		(* Menu war aktiv -> Escape -> Menu deaktivieren *)
	ELSIF (Xus_TN_MENU.in_State = INT#02) THEN
		us_TN_MENU_POPUP.bo_Destroy := TRUE;
		Xus_TN_MENU.bo_Update := TRUE;
		Xus_TN_MENU.in_State := INT#01;
		bo_Reset_Position := TRUE;

		Xus_TN_SCREEN.bo_Menue_Bar_Dialog := FALSE;
	END_IF;
END_IF;

(* Menu aktiv *)
IF (Xus_TN_MENU.in_State = INT#02) THEN

	(* Return *)
	IF (by_New_KeyCode = BYTE#13)  THEN
		us_TN_MENU_POPUP.bo_Destroy := TRUE;
		Xus_TN_MENU.bo_Update := TRUE;
		Xus_TN_MENU.in_State := INT#01;
		bo_Reset_Position := TRUE;
		Xus_TN_MENU.in_Menu_Selected := (Xus_TN_MENU.in_Cur_Menu_Item * INT#10) + Xus_TN_MENU.in_Cur_Sub_Item;
		Xus_TN_SCREEN.by_Input_Exten_Code := BYTE#00;

		Xus_TN_SCREEN.bo_Menue_Bar_Dialog := FALSE;

		(* Destroy-Befehl -> Popup-Menu beenden *)
	ELSIF (Xus_TN_MENU.bo_Destroy = TRUE) THEN
		us_TN_MENU_POPUP.bo_Destroy := TRUE;
		Xus_TN_MENU.bo_Update := TRUE;
		Xus_TN_MENU.in_State := INT#01;
		bo_Reset_Position := TRUE;
		Xus_TN_MENU.in_Menu_Selected := INT#00;
		Xus_TN_SCREEN.by_Input_Exten_Code := BYTE#00;

		Xus_TN_SCREEN.bo_Menue_Bar_Dialog := FALSE;

	END_IF;

	IF (by_New_KeyCode = BYTE#67) THEN (* Cursor rechts *)
		in_Scroll_Offset := INT#1;
		Xus_TN_MENU.bo_Update := TRUE;
		Xus_TN_SCREEN.by_Input_Exten_Code := BYTE#00;

	ELSIF (by_New_KeyCode = BYTE#68) THEN (* Cursor links *)
		in_Scroll_Offset := -1;
		Xus_TN_MENU.bo_Update := TRUE;
		Xus_TN_SCREEN.by_Input_Exten_Code := BYTE#00;
	END_IF;
END_IF;

IF bo_Reset_Position = TRUE THEN
	bo_Reset_Position := FALSE;
	Xus_TN_MENU.in_X_SM_old := -1;
	Xus_TN_MENU.in_Y_SM_old := -1;
	Xus_TN_MENU.in_X_SM_new := -1;
	Xus_TN_MENU.in_Y_SM_new := -1;
END_IF;

(* POPUP-Menu updaten *)
IF (Xus_TN_MENU.in_State > INT#00) AND (Xus_TN_MENU.bo_Update = TRUE) THEN

	Xus_TN_MENU.bo_Update := FALSE; 

	in_ROW := Xus_TN_MENU.in_Y;
	in_COL := Xus_TN_MENU.in_X;

	(* Scrolloffset *)
	IF in_Scroll_Offset <> INT#00 THEN
		Xus_TN_MENU.in_Cur_Menu_Item := INC2(Xus_TN_MENU.in_Cur_Menu_Item,in_Scroll_Offset,1,Xus_TN_MENU.in_Menu_E_Count);
		in_Scroll_Offset := INT#00;
	ELSE
		(* Item = 0 und kein Scrolloffset *)
		IF (Xus_TN_MENU.in_Cur_Menu_Item = INT#00) THEN
			Xus_TN_MENU.in_Cur_Menu_Item := INT#01;
		END_IF;
	END_IF;

	(* alle Menutext zeichnen *)
	FOR in_Count := INT#01 TO Xus_TN_MENU.in_Menu_E_Count DO;

		(* Zeichenfarbe bestimmen *)
		IF (in_Count = Xus_TN_MENU.in_Cur_Menu_Item) AND (Xus_TN_MENU.in_State > INT#01 ) THEN
			by_ATTR := Xus_TN_MENU.by_Attr_mF;

			Xus_TN_MENU.in_Y_SM_new := in_ROW + INT#01;
			Xus_TN_MENU.in_X_SM_new := in_COL;

		ELSE
			by_ATTR := Xus_TN_MENU.by_Attr_oF;
		END_IF;

		st_MENU_TITLE := ELEMENT_GET(SEP:=BYTE#35,POS:=in_Count - 1,ELEMENT:=st_MENU_BAR);

		in_TITLE_Length := LEN(st_MENU_TITLE) + INT#02;

		FB_TN_SC_WRITE_C(	Iin_Y := in_ROW,
							Iin_X := in_COL,
							Iby_ATTR := by_ATTR,
							Iin_LENGTH := in_TITLE_Length,
							Iin_OPTION := INT#02,
							Ist_STRING := st_MENU_TITLE,
							Xus_TN_SCREEN := Xus_TN_SCREEN);

		in_COL := in_COL + in_TITLE_Length;

	END_FOR;
END_IF;

IF Xus_TN_MENU.in_X_SM_new <> Xus_TN_MENU.in_X_SM_old THEN

	(* SubMenu ist aktiv -> beenden                                     *)
	IF us_TN_MENU_POPUP.bo_Activ = TRUE THEN
		us_TN_MENU_POPUP.bo_Destroy := TRUE;

		(* Sub-Menu bearbeiten *)
		FB_TN_INPUT_MENU_POPUP(	Xus_TN_MENU_POPUP := us_TN_MENU_POPUP,
								Xus_TN_SCREEN := Xus_TN_SCREEN);
	END_IF;

	IF us_TN_MENU_POPUP.bo_Activ = FALSE THEN
		(* Popup-Menu zu aktuellen Menu parametrieren und ausführen         *)
		in_Index := Xus_TN_MENU.in_Cur_Menu_Item;

		us_TN_MENU_POPUP.in_Y := Xus_TN_MENU.in_Y_SM_new;
		us_TN_MENU_POPUP.in_X := Xus_TN_MENU.in_X_SM_new;
		us_TN_MENU_POPUP.by_Attr_mF := Xus_TN_MENU.by_Attr_mF;
		us_TN_MENU_POPUP.by_Attr_oF := Xus_TN_MENU.by_Attr_oF;
		us_TN_MENU_POPUP.st_Menu_Text := ELEMENT_GET(SEP:=BYTE#37,POS:=in_Index,ELEMENT:=Xus_TN_MENU.st_MENU_TEXT);
		us_TN_MENU_POPUP.bo_Create := TRUE;

		Xus_TN_MENU.in_X_SM_old := Xus_TN_MENU.in_X_SM_new;
		Xus_TN_MENU.in_Y_SM_old := Xus_TN_MENU.in_Y_SM_new;

	END_IF;
END_IF;

(* Popup-Menu zyklisch aufrufen *)
FB_TN_INPUT_MENU_POPUP(	Xus_TN_MENU_POPUP := us_TN_MENU_POPUP,
						Xus_TN_SCREEN := Xus_TN_SCREEN);

(* aktuelles Item vom Popup-Menu kopieren *)
Xus_TN_MENU.in_Cur_Sub_Item := us_TN_MENU_POPUP.in_Cur_Item;

(* Destroy-Befehl *)
IF (Xus_TN_MENU.in_State = INT#01) THEN
	IF (Xus_TN_MENU.bo_Destroy = TRUE) THEN
		Xus_TN_MENU.in_State := INT#00;
		Xus_TN_MENU.bo_Destroy := FALSE;
		Xus_TN_MENU.in_Cur_Menu_Item := INT#00;
		Xus_TN_MENU.in_Cur_Sub_Item := INT#00;
	END_IF;
END_IF;

(* revision history
ks	06. apr. 2011	rev 1.1
	list_len und list_get durch element_count und element_get ersetzt

ks	10. mai. 2010	rev 1.0
	original version
*)

END_FUNCTION_BLOCK

// ---- POUs/TELNET_VISION/TN_RECEIVE.TcPOU
FUNCTION_BLOCK TN_RECEIVE
VAR_IN_OUT
	R_BUF :	NETWORK_BUFFER;
	Xus_TN_SCREEN : us_TN_SCREEN;
END_VAR
VAR
	REQ_Size : UINT;
	REQ1 : BYTE;
	REQ2 : BYTE;
	REQ3 : BYTE;
END_VAR

(*
version 1.0		10. mai 2010
programmer		ks
tested by		ks

TN_RECEIVE empfängt Tastatureingaben vom Telnet Client und wertet diese aus
*)

(* Datenempfang auswertung *)
Xus_TN_SCREEN.by_Input_ASCII_Code := BYTE#00;
Xus_TN_SCREEN.by_Input_Exten_Code := BYTE#00;

IF R_BUF.SIZE > UINT#0 THEN
	(* empfangene Daten auswerten *)
	REQ_Size := R_BUF.SIZE;
	REQ1 := R_BUF.BUFFER[0];
	REQ2 := R_BUF.BUFFER[1];
	REQ3 := R_BUF.BUFFER[2];

	IF REQ1 = BYTE#27 AND REQ_Size >= UINT#3 THEN (* Escape *)
		IF REQ2 = BYTE#91 THEN (* Cursor code *)
			IF (REQ3 >= BYTE#65 AND REQ3 <= BYTE#68) OR (REQ3 = BYTE#72) OR (REQ3 = BYTE#75) THEN (* 65..68 = Cursor o,u,r,l / 72 = POS1 / 75 = ENDE *)
				Xus_TN_SCREEN.by_Input_Exten_Code := REQ3;
			END_IF;
		ELSIF REQ2 = BYTE#79 THEN (* Sondertasten F1/F2/F3/F4 *)
			IF REQ3 >= BYTE#80 AND REQ3 <= BYTE#83 THEN
				Xus_TN_SCREEN.by_Input_Exten_Code := REQ3;
			END_IF;
		END_IF;
	ELSIF REQ1 >= BYTE#32 AND REQ1 <= BYTE#126 THEN
		Xus_TN_SCREEN.by_Input_ASCII_Code := REQ1;
		Xus_TN_SCREEN.bo_Input_ASCII_IsNum := ISC_NUM(REQ1); (* Auswertung auf Zahleneingabe *)
	ELSIF REQ1 = BYTE#8 OR REQ1 = BYTE#9 OR REQ1 = BYTE#13 OR REQ1 = BYTE#27 THEN (* prüfe auf Steuerzeichen 8=Backspace / 9=Tabulator / 13=Return / 27=Escape *)
		Xus_TN_SCREEN.by_Input_Exten_Code := REQ1;
	END_IF;

	(* Empfangsbuffer Datenlänge null eintragen (Telegramm zerstören *)
	R_BUF.SIZE := UINT#00;
END_IF;

(* revision history
ks	10. mai. 2010	rev 1.0
	original version
*)

END_FUNCTION_BLOCK

// ---- POUs/TELNET_VISION/TN_SEND_ROWS.TcPOU
FUNCTION_BLOCK TN_SEND_ROWS
VAR_IN_OUT
	IP_C : IP_C;
	S_BUF : NETWORK_BUFFER;
	Xus_TN_SCREEN : us_TN_SCREEN;
END_VAR
VAR_INPUT
	S_BUF_SIZE : INT;
END_VAR
VAR
	in_Line_Count : INT;(*Zähler um max alle 24 Zeilen zu durchlaufen*)
	in_Col_Count : INT;
	in_Last_Row_Index : INT;
	bo_Break_Loop : BOOL;
	in_Row_Count : INT;
	in_Offset : INT;
	in_Write_Index : INT;
	in_Write_Index_Backup : INT;
	by_Cur_Color : BYTE;
	by_last_Color : BYTE;
	in_Write_Stop : INT;
END_VAR

(*
version 1.0		10. mai 2010
programmer		ks
tested by		ks

TN_SEND_ROWS prüft den Bildschirmspeicher auf änderungen, und sendet diese zeilenweise an den Telnet Client 
*)

(* Verbindung vorhanden und kein Datensenden aktiv *)
IF (IP_C.C_STATE < BYTE#127 OR S_BUF.SIZE > UINT#0) THEN
	RETURN; (* nein -> Baustein beenden *)
END_IF;

(* aktuellen Schreibindex laden *)
in_Write_Index := UINT_TO_INT(S_BUF.SIZE) - 1;

(* aktuellen Schreibindex zwischenspeichern *)
in_Write_Index_Backup := in_Write_Index;

(* positive Flanke Connect on *)
IF (IP_C.C_STATE = BYTE#254) OR (Xus_TN_SCREEN.bo_Clear_Screen) THEN

	(* Clear-Screen Meldung rücksetzen *)
	Xus_TN_SCREEN.bo_Clear_Screen := FALSE;

	(* alle Zeilen für Update markieren *)
	FOR in_Line_Count := INT#00 TO INT#23 DO
		Xus_TN_SCREEN.bya_Line_Update[in_Line_Count] := TRUE;
	END_FOR;

	(* ESC [0;30,40m  Reset Attributes + Black,Black *)
	in_Write_Index := in_Write_Index + INT#1;
	S_BUF.BUFFER[in_Write_Index] := BYTE#16#1B; (* ESC *)
	in_Write_Index := in_Write_Index + INT#1;
	S_BUF.BUFFER[in_Write_Index] := BYTE#16#5B; (* [ *)
	in_Write_Index := in_Write_Index + INT#1;
	S_BUF.BUFFER[in_Write_Index] := BYTE#16#30; (* 0 *)
	in_Write_Index := in_Write_Index + INT#1;
	S_BUF.BUFFER[in_Write_Index] := BYTE#16#3B; (* ; *)
	in_Write_Index := in_Write_Index + INT#1;
	S_BUF.BUFFER[in_Write_Index] := BYTE#16#33; (* 3 *)

	(* Einerstelle Farbe Foreground ausgeben *)
	in_Write_Index := in_Write_Index + INT#1;
	S_BUF.BUFFER[in_Write_Index] := (SHR(Xus_TN_SCREEN.by_Clear_Screen_Attr,4) OR BYTE#16#30);

	in_Write_Index := in_Write_Index + INT#1;
	S_BUF.BUFFER[in_Write_Index] := BYTE#16#3B; (* ; *)
	in_Write_Index := in_Write_Index + INT#1;
	S_BUF.BUFFER[in_Write_Index] := BYTE#16#34; (* 4 *)

	(* Einerstelle Farbe Background ausgeben *)
	in_Write_Index := in_Write_Index + INT#1;
	S_BUF.BUFFER[in_Write_Index] := ((Xus_TN_SCREEN.by_Clear_Screen_Attr AND BYTE#16#07) OR BYTE#16#30);

	in_Write_Index := in_Write_Index + INT#1;
	S_BUF.BUFFER[in_Write_Index] := BYTE#16#6D; (* m *)

	(* ESC[2J Clear screen and home cursor *)
	in_Write_Index := in_Write_Index + INT#1;
	S_BUF.BUFFER[in_Write_Index] := BYTE#16#1B; (* ESC *)
	in_Write_Index := in_Write_Index + INT#1;
	S_BUF.BUFFER[in_Write_Index] := BYTE#16#5B; (* [ *)
	in_Write_Index := in_Write_Index + INT#1;
	S_BUF.BUFFER[in_Write_Index] := BYTE#16#32; (* 2 *)
	in_Write_Index := in_Write_Index + INT#1;
	S_BUF.BUFFER[in_Write_Index] := BYTE#16#4A; (* J *)

	(* ESC [?7l Off *)
	in_Write_Index := in_Write_Index + INT#1;
	S_BUF.BUFFER[in_Write_Index] := BYTE#16#1B; (* ESC *)
	in_Write_Index := in_Write_Index + INT#1;
	S_BUF.BUFFER[in_Write_Index] := BYTE#16#5B; (* [ *)
	in_Write_Index := in_Write_Index + INT#1;
	S_BUF.BUFFER[in_Write_Index] := BYTE#16#3F; (* ? *)
	in_Write_Index := in_Write_Index + INT#1;
	S_BUF.BUFFER[in_Write_Index] := BYTE#16#37; (* 7 *)
	in_Write_Index := in_Write_Index + INT#1;
	S_BUF.BUFFER[in_Write_Index] := BYTE#16#6C; (* l *)

END_IF;

in_Last_Row_Index := INT#0;
bo_Break_Loop := FALSE;
in_Write_Stop := S_BUF_SIZE - 20;

(* alle Zeilen durchlaufen *)
FOR in_Line_Count := 0 TO 23 DO

	in_Offset := in_Row_Count * INT#80;

	(* prüfen ob Update einer Zeile notwendig ist bzw. nach Reconnect *)
	IF (Xus_TN_SCREEN.bya_Line_Update[in_Row_Count] = TRUE) THEN

		(* Schreib-Cursor positionieren *)
		in_Write_Index := in_Write_Index + INT#1;
		S_BUF.BUFFER[in_Write_Index] := BYTE#16#1B; (* ESC *)
		in_Write_Index := in_Write_Index + INT#1;
		S_BUF.BUFFER[in_Write_Index] := BYTE#16#5B; (* [ *)

		(* Zehnerstelle Zeilennummer ausgeben *)
		in_Write_Index := in_Write_Index + INT#1;
		S_BUF.BUFFER[in_Write_Index] :=
		SHR(INT_TO_BCDC(in_Row_Count + INT#1),INT#4) OR BYTE#16#30;

		(* Einerstelle Zeilennummer ausgeben *)
		in_Write_Index := in_Write_Index + INT#1;
		S_BUF.BUFFER[in_Write_Index] :=
		(INT_TO_BCDC(in_Row_Count + INT#1) AND BYTE#16#0F) OR BYTE#16#30;

		in_Write_Index := in_Write_Index + INT#1;
		S_BUF.BUFFER[in_Write_Index] := BYTE#16#3B; (* ; *)
		in_Write_Index := in_Write_Index + INT#1;
		S_BUF.BUFFER[in_Write_Index] := BYTE#16#31; (* 1 *)
		in_Write_Index := in_Write_Index + INT#1;
		S_BUF.BUFFER[in_Write_Index] := BYTE#16#48; (* H *)

		(* alle Spalten einer Zeile durchlaufen *)
		FOR in_Col_Count := 0 TO 79 DO

			(* aktuelle Farbe bestimmen *)
			by_Cur_Color := Xus_TN_SCREEN.bya_COLOR[in_Offset];
			IF (by_Cur_Color <> by_last_Color) OR (in_Col_Count = INT#00) THEN

				(* Farbeinstellung: ANSI-Sequenz ESC[X;Y;Zm ausgeben *)
				in_Write_Index := in_Write_Index + INT#1;
				S_BUF.BUFFER[in_Write_Index] := BYTE#16#1B; (* ESC *)

				in_Write_Index := in_Write_Index + INT#1;
				S_BUF.BUFFER[in_Write_Index] := BYTE#16#5B; (* [ *)

				(* Farbeinstellung: dunkel oder Hell und blinken bestimmen *)

					IF (((by_Cur_Color AND BYTE#2#10001000) XOR (by_last_Color AND BYTE#2#10001000)) <> BYTE#00) OR (in_Col_Count = 0) THEN

						in_Write_Index := in_Write_Index + INT#1;
						S_BUF.BUFFER[in_Write_Index] := BYTE#16#30; (* 0 *)
						in_Write_Index := in_Write_Index + INT#1;
						S_BUF.BUFFER[in_Write_Index] := BYTE#16#3B; (* ; *)

						(* keine dunklen Farben gewünscht -> dann Bold & Bright *)
						IF (by_Cur_Color AND BYTE#2#00001000) = BYTE#2#00000000 THEN

							(* auf Bold & Btight Farben umstellen *)
							in_Write_Index := in_Write_Index + INT#1;
							S_BUF.BUFFER[in_Write_Index] := BYTE#16#31; (* 1 *) 
							in_Write_Index := in_Write_Index + INT#1;
							S_BUF.BUFFER[in_Write_Index] := BYTE#16#3B; (* ; *)

						END_IF;

						(* blinkenden Farben gewünscht *)
						IF (by_Cur_Color AND BYTE#2#10000000) = BYTE#2#10000000 THEN 

							(* auf Bold & Bright Farben umstellen *)
							in_Write_Index := in_Write_Index + INT#1;
							S_BUF.BUFFER[in_Write_Index] := BYTE#16#35; (* 5 *) 
							in_Write_Index := in_Write_Index + INT#1;
							S_BUF.BUFFER[in_Write_Index] := BYTE#16#3B; (* ; *)

						END_IF;

					END_IF;

					(* Zehnerstelle Farbe Foreground ausgeben *)
					in_Write_Index := in_Write_Index + INT#1;
					S_BUF.BUFFER[in_Write_Index] := BYTE#16#33; (* 3 *)

					(* Einerstelle Farbe Foreground ausgeben *)
					in_Write_Index := in_Write_Index + INT#1;
					S_BUF.BUFFER[in_Write_Index] := ((SHR(by_Cur_Color,4) AND BYTE#2#00000111) OR BYTE#16#30);

					in_Write_Index := in_Write_Index + INT#1;
					S_BUF.BUFFER[in_Write_Index] := BYTE#16#3B; (* ; *)

					(* Zehnerstelle Farbe Background ausgeben *)
					in_Write_Index := in_Write_Index + INT#1;
					S_BUF.BUFFER[in_Write_Index] := BYTE#16#34; (* 4 *)

					(* Einerstelle Farbe Background ausgeben *)
					in_Write_Index := in_Write_Index + INT#1;
					S_BUF.BUFFER[in_Write_Index] := ((by_Cur_Color AND BYTE#2#00000111) OR BYTE#16#30); 

					in_Write_Index := in_Write_Index + INT#1;
					S_BUF.BUFFER[in_Write_Index] := BYTE#16#6D; (* m *)

					(* neue Farbe als letzt verwendete speichern *)
					by_last_Color := by_Cur_Color;

				END_IF;

				(* Buffer Ende vorzeitig erreicht -> Ende *)
				IF (in_Write_Index > in_Write_Stop) THEN

					bo_Break_Loop := TRUE;
					EXIT;

				END_IF;

				(* ein TEXT-Zeichen von Screenbuffer in den Sendebuffer übertragen *)
				in_Write_Index := in_Write_Index + INT#1;
				S_BUF.BUFFER[in_Write_Index] := Xus_TN_SCREEN.bya_CHAR[in_Offset];

				(* nächste Spalte anwählen *)
				in_Offset := in_Offset + INT#01;
			END_FOR;

			IF (bo_Break_Loop = TRUE) THEN;

				(* Buffer Ende vorzeitig erreicht -> nur bis zur letzten kompletten Zeile uebertragen *)
				in_Write_Index := in_Last_Row_Index;

				EXIT;
			END_IF;

			(* Buffer ist noch nicht voll -> neue Zeile ubernehmen *)
			in_Last_Row_Index := in_Write_Index;
			Xus_TN_SCREEN.bya_Line_Update[in_Row_Count] := FALSE;

		END_IF;

		(* naechste Zeile adressieren *)
		in_Row_Count := in_Row_Count + INT#01;

		(* ab letzter Zeile wieder von vorne beginnen *)
		IF (in_Row_Count > INT#23) THEN
			in_Row_Count := INT#00;
		END_IF;
		(*-----------------------------------------------*)


	END_FOR;

	(* wenn in einen Update-Zyklus alle Zeilen auf einmal geschafft wurden *)
	(* wird der Row_Count auf ersten Zeile gestellt *)
	(* soll das hässliche Grafikflackern verhindern *)
	(* ansonsten wird bei der letzen Zeile weitergemacht *)
	IF (bo_Break_Loop = FALSE) THEN
		in_Row_Count := INT#00;
	END_IF;

	(* Edit-Cursor positionieren *)
	IF (in_Write_Index <> in_Write_Index_Backup) THEN

		in_Write_Index := in_Write_Index + INT#1;
		S_BUF.BUFFER[in_Write_Index] := BYTE#16#1B; (* ESC *)
		in_Write_Index := in_Write_Index + INT#1;
		S_BUF.BUFFER[in_Write_Index] := BYTE#16#5B; (* [ *)

		(* Zehnerstelle Zeilennummer ausgeben *)
		in_Write_Index := in_Write_Index + INT#1;
		S_BUF.BUFFER[in_Write_Index] := SHR(INT_TO_BCDC(Xus_TN_SCREEN.in_Cursor_Y + 1),INT#4) OR BYTE#16#30;

		(* Einerstelle Zeilennummer ausgeben *)
		in_Write_Index := in_Write_Index + INT#1;
		S_BUF.BUFFER[in_Write_Index] := (INT_TO_BCDC(Xus_TN_SCREEN.in_Cursor_Y + 1) AND BYTE#16#0F) OR BYTE#16#30;

		in_Write_Index := in_Write_Index + INT#1;
		S_BUF.BUFFER[in_Write_Index] := BYTE#16#3B; (* ; *)

		(* Zehnerstelle Spaltenummer ausgeben *)
		in_Write_Index := in_Write_Index + INT#1;
		S_BUF.BUFFER[in_Write_Index] := SHR(INT_TO_BCDC(Xus_TN_SCREEN.in_Cursor_X + 1),INT#4) OR BYTE#16#30;

		(* Einerstelle Spaltennummer ausgeben *)
		in_Write_Index := in_Write_Index + INT#1;
		S_BUF.BUFFER[in_Write_Index] := (INT_TO_BCDC(Xus_TN_SCREEN.in_Cursor_X + 1) AND BYTE#16#0F) OR BYTE#16#30;

		in_Write_Index := in_Write_Index + INT#1;
		S_BUF.BUFFER[in_Write_Index] := BYTE#16#48; (* H *)

END_IF;

(* aktuellen Schreibindex speichern -> Senden anstossen *)
S_BUF.SIZE := TO_UINT(in_Write_Index + 1);

(* revision history
ks	10. mai. 2010	rev 1.0
	original version
*)

END_FUNCTION_BLOCK

// ---- POUs/NETWORK/LOG_VIEWPORT.TcPOU
FUNCTION_BLOCK LOG_VIEWPORT
VAR_IN_OUT
	LC : LOG_CONTROL;
	LV : us_LOG_VIEWPORT;
END_VAR
VAR
	pos : INT;
	count : INT;
	idx : INT;
	base : INT;
	update_pos : BOOL;
END_VAR

(*
version 1.0		01 mai 2010
programmer		ks
tested BY		ks

LOG_VIEWPORT erzeugt einen Liste der Meldungen des Loggingbuffers die innerhalb einer virtuellen Ansicht enthalten sind.
*)

(* Scroll Button verarbeiten *)
IF LV.MOVE_TO_X <> 0 THEN
	CASE LV.MOVE_TO_X OF
	30000: pos := 1 ; (* älteste Meldung anzeigen *)
	30001: pos := LC.SIZE; (* neueste Meldung anzeigen *)
	30002: pos := pos + LV.COUNT; (* eine Seite nach unten blättern -> Richtung neuere Nachrichten *)
	30003: pos := pos - LV.COUNT; (* eine Seite nach oben blättern -> Richtung ältere Nachrichten *)
	ELSE
		pos := pos + LV.MOVE_TO_X;
	END_CASE;
	update_pos := TRUE;
	LV.MOVE_TO_X := 0;
END_IF;

IF (LV.UPDATE_COUNT <> LC.UPDATE_COUNT) OR update_pos THEN (* Aktualisierung überwachen *)
	LV.UPDATE := TRUE;
	LV.UPDATE_COUNT := LC.UPDATE_COUNT;
	update_pos := FALSE;

	(* pos prüfen und übernehmen *)
	IF LC.RING_MODE THEN
		pos := LIMIT(1,pos,LC.SIZE - LV.COUNT + 1);
	ELSE
		IF LC.IDX > LV.COUNT THEN
			pos := LIMIT(1,pos,LC.IDX - LV.COUNT + 1);
		ELSE
			pos := 1;
		END_IF;
	END_IF;

	(* idxBasis berechnen *)
	base := LC.IDX - pos - LV.COUNT + 1;
	IF LC.RING_MODE THEN 
		(* Anzeige im Ringpuffermodus *)
		FOR count:= 1 TO LV.COUNT DO
			idx := base + count;
			IF idx < 1 THEN
				idx := idx + LC.SIZE;
			END_IF;
		END_FOR;
	ELSE
		(* Anzeige im Normalmodus *)
		FOR count:= 1 TO LV.COUNT DO
			idx := base + count;
			IF idx < 1 THEN
				(* Leere Zeile ausgeben *)
				LV.LINE_ARRAY[count] := 0;
			ELSE
				LV.LINE_ARRAY[count] := idx;
			END_IF;
		END_FOR;
	END_IF;
END_IF;

(* revision history
ks	01. mai 2010	rev 1.0
	original version
*)

END_FUNCTION_BLOCK

// ---- POUs/TELNET_VISION/TN_SC_VIEWPORT.TcPOU
FUNCTION_BLOCK TN_SC_VIEWPORT
VAR
	FB_TN_SC_WRITE : TN_SC_WRITE;
	FB_TON : TON;
END_VAR
VAR
	in_index : INT;
	in_Color : INT;
	by_Attr : BYTE;
	in_count : INT;
END_VAR
VAR_IN_OUT
	Xus_LOG_VIEWPORT : us_LOG_VIEWPORT;
	Xus_LOG_CONTROL : LOG_CONTROL;
	Xus_TN_SCREEN : us_TN_SCREEN;
END_VAR
VAR_INPUT
	Iin_X : INT;
	Iin_Y : INT;
	Iin_Width : INT;
	Idw_ATTR_1 : DWORD;
	Idw_ATTR_2 : DWORD;
	Iti_TIME : TIME;
END_VAR

(*
version 1.0		10. mai 2010
programmer		ks
tested by		ks

TN_SC_VIEWPORT verwaltet und zeichnet einen rechteckigen Bereich in dem der Log-buffer angezeigt wird
*)

(* LOG-Messages ausgeben *)

IF Xus_LOG_VIEWPORT.UPDATE AND FB_TON.Q THEN (* Update gewünscht und Verzögerungszeit abgelaufen *)
	Xus_LOG_VIEWPORT.UPDATE := FALSE;
	FOR in_count := 1 TO Xus_LOG_VIEWPORT.COUNT DO (* Alle Viewport-Zeilen abarbeiten *)
		in_index := Xus_LOG_VIEWPORT.LINE_ARRAY[in_count];
		(* Farbe aus den Option-Parameter auslesen >0,Level,Back,Front< *)
		in_Color := DWORD_TO_INT(Xus_LOG_CONTROL.MSG_OPTION[in_index] AND DWORD#2#1111);

		CASE in_Color OF
		0..3: by_Attr := BYTE_OF_DWORD(Idw_ATTR_1,INT_TO_BYTE(in_Color));
		4..7: by_Attr := BYTE_OF_DWORD(Idw_ATTR_2,INT_TO_BYTE(in_Color));
		ELSE
			by_Attr := BYTE_OF_DWORD(Idw_ATTR_1,BYTE#0);
		END_CASE;

		(* Message (Text + Farbe) ausgeben *)
		FB_TN_SC_WRITE(	Iin_Y := Iin_Y + in_count - INT#01,
						Iin_X := Iin_X,
						Iby_ATTR := by_Attr,
						Ist_STRING := FIX(str := Xus_LOG_CONTROL.MSG[in_index], L := Iin_Width, C := BYTE#32, M := INT#00), (* String rechts ergänzen bzw. kürzen *)
						Xus_TN_SCREEN := Xus_TN_SCREEN);

	END_FOR;

	(* Timer stoppen/rücksetzen *)
	FB_TON.IN := FALSE;
	FB_TON.PT := Iti_TIME;
	FB_TON();

END_IF;

(* Update-Zeitverzoegerung *)
FB_TON.IN := TRUE;
FB_TON.PT := Iti_TIME;
FB_TON();

(* revision history
ks	10. mai. 2010	rev 1.0
	original version
*)

END_FUNCTION_BLOCK

// ---- POUs/DEMO/TN_VISION_DEMO_2.TcPOU
PROGRAM TN_VISION_DEMO_2
VAR
	FB_TN_FRAMEWORK : TN_FRAMEWORK;
	FB_TN_SC_FILL : TN_SC_FILL;
	FB_TN_SC_WRITE_C : TN_SC_WRITE_C;
	FB_TN_SC_WRITE : TN_SC_WRITE;
	Xus_TN_MENU : us_TN_MENU;
	Xus_TN_INPUT_CONTROL : us_TN_INPUT_CONTROL;
	Xus_TN_SCREEN : us_TN_SCREEN;
	S_BUF : NETWORK_BUFFER;
	R_BUF : NETWORK_BUFFER;
	IP_C : IP_C;
END_VAR

FB_TN_FRAMEWORK(
	us_TN_INPUT_CONTROL := Xus_TN_INPUT_CONTROL ,
	us_TN_SCREEN := Xus_TN_SCREEN ,
	us_TN_MENU := Xus_TN_MENU ,
	S_BUF := S_BUF ,
	R_BUF:= R_BUF ,
	IP_C:= IP_C );

(* Initialisierung der Daten und Strukturen *)
IF (Xus_TN_SCREEN.in_Page_Number = INT#00) THEN
	Xus_TN_SCREEN.in_Page_Number := INT#01;

	(* Clear-Screen (Farbe setzen + Display löschen) *)
	Xus_TN_SCREEN.by_Clear_Screen_Attr := BYTE#16#00;
	Xus_TN_SCREEN.bo_Clear_Screen := TRUE;

	(* Screen initialisieren (mit Leerzeichen füllen) *)
	FB_TN_SC_FILL(	Iin_X1 := INT#00,
					Iin_Y1 := INT#00,
					Iin_X2 := INT#79,
					Iin_Y2 := INT#23,
					Iby_CHAR := BYTE#32,
					Iby_Attr := BYTE#16#00,
					Xus_TN_SCREEN := Xus_TN_SCREEN);

	(* Statische Texte ausgeben *)
	FB_TN_SC_WRITE(	Iin_X := INT#00,
					Iin_Y := INT#00,
					Iby_ATTR := BYTE#16#70,
					Ist_STRING := 'Login Screen                                                     FL SWITCH MM HS',
					Xus_TN_SCREEN := Xus_TN_SCREEN);

	(* Statische Texte ausgeben *)
	FB_TN_SC_WRITE(	Iin_X := INT#00,
					Iin_Y := INT#03,
					Iby_ATTR := BYTE#16#70,
					Ist_STRING := 'XXXXXXXXX',
					Xus_TN_SCREEN := Xus_TN_SCREEN);

	(* Statische Texte ausgeben *)
	FB_TN_SC_WRITE(	Iin_X := INT#00,
					Iin_Y := INT#04,
					Iby_ATTR := BYTE#16#70,
					Ist_STRING := 'X   X  XX',
					Xus_TN_SCREEN := Xus_TN_SCREEN);

	(* Statische Texte ausgeben *)
	FB_TN_SC_WRITE(	Iin_X := INT#00,
					Iin_Y := INT#05,
					Iby_ATTR := BYTE#16#70,
					Ist_STRING := 'X   O   X      ---> Phoenix Contact Managed Switch System <---',
					Xus_TN_SCREEN := Xus_TN_SCREEN);

	(* Statische Texte ausgeben *)
	FB_TN_SC_WRITE(	Iin_X := INT#00,
					Iin_Y := INT#06,
					Iby_ATTR := BYTE#16#70,
					Ist_STRING := 'X   X  XX               Phoenix Contact GmbH & Co KG',
					Xus_TN_SCREEN := Xus_TN_SCREEN);

	(* Statische Texte ausgeben *)
	FB_TN_SC_WRITE(	Iin_X := INT#00,
					Iin_Y := INT#07,
					Iby_ATTR := BYTE#16#70,
					Ist_STRING := 'X   XXXXX                   www.PhoenixContact.com',
					Xus_TN_SCREEN := Xus_TN_SCREEN);

	(* Statische Texte ausgeben *)
	FB_TN_SC_WRITE(	Iin_X := INT#00,
					Iin_Y := INT#08,
					Iby_ATTR := BYTE#16#70,
					Ist_STRING := 'X   XXXXX',
					Xus_TN_SCREEN := Xus_TN_SCREEN);

	(* Statische Texte ausgeben *)
	FB_TN_SC_WRITE(	Iin_X := INT#00,
					Iin_Y := INT#09,
					Iby_ATTR := BYTE#16#70,
					Ist_STRING := 'XXXXXXXXX',
					Xus_TN_SCREEN := Xus_TN_SCREEN);

	(* Statische Texte ausgeben *)
	FB_TN_SC_WRITE(	Iin_X := INT#00,
					Iin_Y := INT#11,
					Iby_ATTR := BYTE#16#70,
					Ist_STRING := '                Running switch application version:  4.00',
					Xus_TN_SCREEN := Xus_TN_SCREEN);

	(* Alle Input-Controls initialisieren *)

	Xus_TN_INPUT_CONTROL.bo_Enable := FALSE;

  (* Initialisierung der Eingabe-Zeile *)
	Xus_TN_INPUT_CONTROL.usa_TN_INPUT_CONTROL_DATA[1].in_Type := INT#01;
	Xus_TN_INPUT_CONTROL.usa_TN_INPUT_CONTROL_DATA[1].in_Y := INT#17;
	Xus_TN_INPUT_CONTROL.usa_TN_INPUT_CONTROL_DATA[1].in_X := INT#33;
	Xus_TN_INPUT_CONTROL.usa_TN_INPUT_CONTROL_DATA[1].by_Attr_mF := BYTE#16#70;
	Xus_TN_INPUT_CONTROL.usa_TN_INPUT_CONTROL_DATA[1].by_Attr_oF := BYTE#16#70;
	Xus_TN_INPUT_CONTROL.usa_TN_INPUT_CONTROL_DATA[1].in_Cursor_Pos := INT#0;
	Xus_TN_INPUT_CONTROL.usa_TN_INPUT_CONTROL_DATA[1].bo_Input_Only_Num := FALSE;
	Xus_TN_INPUT_CONTROL.usa_TN_INPUT_CONTROL_DATA[1].bo_Input_Hidden := TRUE;
	Xus_TN_INPUT_CONTROL.usa_TN_INPUT_CONTROL_DATA[1].st_Input_Mask := '                ';
	Xus_TN_INPUT_CONTROL.usa_TN_INPUT_CONTROL_DATA[1].st_Input_Data := Xus_TN_INPUT_CONTROL.usa_TN_INPUT_CONTROL_DATA[1].st_Input_Mask;
	Xus_TN_INPUT_CONTROL.usa_TN_INPUT_CONTROL_DATA[1].st_Input_ToolTip := '';
	Xus_TN_INPUT_CONTROL.usa_TN_INPUT_CONTROL_DATA[1].in_Input_Option := INT#00;
	Xus_TN_INPUT_CONTROL.usa_TN_INPUT_CONTROL_DATA[1].in_Title_Y_Offset := INT#00;
	Xus_TN_INPUT_CONTROL.usa_TN_INPUT_CONTROL_DATA[1].in_Title_X_Offset := -12;
	Xus_TN_INPUT_CONTROL.usa_TN_INPUT_CONTROL_DATA[1].by_Title_Attr := BYTE#16#70;
	Xus_TN_INPUT_CONTROL.usa_TN_INPUT_CONTROL_DATA[1].st_Title_String := 'Password:  [                ]';

	(* Control-Tool-Tip *)
	Xus_TN_INPUT_CONTROL.in_ToolTip_Y := INT#23;
	Xus_TN_INPUT_CONTROL.in_ToolTip_X := INT#09;
	Xus_TN_INPUT_CONTROL.by_ToolTip_Attr := BYTE#16#70;
	Xus_TN_INPUT_CONTROL.in_ToolTip_Size := INT#30;

	(* Control-Verwaltung initialisieren *)
	Xus_TN_INPUT_CONTROL.in_Count := INT#01;
	Xus_TN_INPUT_CONTROL.bo_Enable := TRUE;
	Xus_TN_INPUT_CONTROL.bo_Reset_Fokus := TRUE;
END_IF;

IF (Xus_TN_SCREEN.in_Page_Number = INT#01) THEN

	(* eingegebenen String übernehmen *)
	IF Xus_TN_INPUT_CONTROL.usa_TN_INPUT_CONTROL_DATA[1].bo_Input_Entered = TRUE THEN

		Xus_TN_INPUT_CONTROL.usa_TN_INPUT_CONTROL_DATA[1].bo_Input_Entered := FALSE;

		Xus_TN_INPUT_CONTROL.usa_TN_INPUT_CONTROL_DATA[1].st_Input_String :=
			LOWERCASE(str:=Xus_TN_INPUT_CONTROL.usa_TN_INPUT_CONTROL_DATA[1].st_Input_String);

		IF Xus_TN_INPUT_CONTROL.usa_TN_INPUT_CONTROL_DATA[1].st_Input_String = 'oscat' THEN
			Xus_TN_SCREEN.in_Page_Number := INT#04;

		ELSE
			FB_TN_SC_WRITE_C(	Iin_Y := Xus_TN_INPUT_CONTROL.in_ToolTip_Y,
								Iin_X := Xus_TN_INPUT_CONTROL.in_ToolTip_X,
								Iby_ATTR := BYTE#16#F1,
								Iin_OPTION := INT#02, (* Center-String *)
								Iin_LENGTH := Xus_TN_INPUT_CONTROL.in_ToolTip_Size,
								Ist_STRING := ' User Password Failed   ',
								Xus_TN_SCREEN := Xus_TN_SCREEN);
		END_IF;
	END_IF;
END_IF;

(* Initialisierung der Daten und Strukturen *)
IF (Xus_TN_SCREEN.in_Page_Number = INT#04) THEN
	Xus_TN_SCREEN.in_Page_Number := INT#05;

	(* Clear-Screen (Farbe setzen + Display löschen) *)
	Xus_TN_SCREEN.by_Clear_Screen_Attr := BYTE#16#00;
	Xus_TN_SCREEN.bo_Clear_Screen := TRUE;

	(* Screen initialisieren (mit Leerzeichen füllen) *)
	FB_TN_SC_FILL(	Iin_X1 := INT#00,
					Iin_Y1 := INT#00,
					Iin_X2 := INT#79,
					Iin_Y2 := INT#23,
					Iby_CHAR := BYTE#32,
					Iby_Attr := BYTE#16#00,
					Xus_TN_SCREEN := Xus_TN_SCREEN);

	(* Statische Texte ausgeben *)
	FB_TN_SC_WRITE(	Iin_X := INT#00,
					Iin_Y := INT#00,
					Iby_ATTR := BYTE#16#70,
					Ist_STRING := 'Basic Switch Configuration                                       FL SWITCH MM HS',
					Xus_TN_SCREEN := Xus_TN_SCREEN);

	(* Statische Texte ausgeben                                         *)
	FB_TN_SC_WRITE(	Iin_X := INT#00,
					Iin_Y := INT#03,
					Iby_ATTR := BYTE#16#70,
					Ist_STRING := 'XXXXXXXXX        MAC Address             : 00:A0:45:00:6E:9B',
					Xus_TN_SCREEN := Xus_TN_SCREEN);

	(* Statische Texte ausgeben *)
	FB_TN_SC_WRITE(	Iin_X := INT#00,
					Iin_Y := INT#04,
					Iby_ATTR := BYTE#16#70,
					Ist_STRING := 'X   X  XX',
					Xus_TN_SCREEN := Xus_TN_SCREEN);

	(* Statische Texte ausgeben *)
	FB_TN_SC_WRITE(	Iin_X := INT#00,
					Iin_Y := INT#05,
					Iby_ATTR := BYTE#16#70,
					Ist_STRING := 'X   O   X',
					Xus_TN_SCREEN := Xus_TN_SCREEN);

	(* Statische Texte ausgeben *)
	FB_TN_SC_WRITE(	Iin_X := INT#00,
					Iin_Y := INT#06,
					Iby_ATTR := BYTE#16#70,
					Ist_STRING := 'X   X  XX',
					Xus_TN_SCREEN := Xus_TN_SCREEN);

	(* Statische Texte ausgeben *)
	FB_TN_SC_WRITE(	Iin_X := INT#00,
					Iin_Y := INT#07,
					Iby_ATTR := BYTE#16#70,
					Ist_STRING := 'X   XXXXX',
					Xus_TN_SCREEN := Xus_TN_SCREEN);

	(* Statische Texte ausgeben *)
	FB_TN_SC_WRITE(	Iin_X := INT#00,
					Iin_Y := INT#08,
					Iby_ATTR := BYTE#16#70,
					Ist_STRING := 'X   XXXXX',
					Xus_TN_SCREEN := Xus_TN_SCREEN);

	(* Statische Texte ausgeben *)
	FB_TN_SC_WRITE(	Iin_X := INT#00,
					Iin_Y := INT#09,
					Iby_ATTR := BYTE#16#70,
					Ist_STRING := 'XXXXXXXXX',
					Xus_TN_SCREEN := Xus_TN_SCREEN);

	(* Alle Input-Controls initialisieren *)

	Xus_TN_INPUT_CONTROL.bo_Enable      := FALSE;

	Xus_TN_INPUT_CONTROL.usa_TN_INPUT_CONTROL_DATA[1].in_Type := INT#01;
	Xus_TN_INPUT_CONTROL.usa_TN_INPUT_CONTROL_DATA[1].in_Y := INT#04;
	Xus_TN_INPUT_CONTROL.usa_TN_INPUT_CONTROL_DATA[1].in_X := INT#44;
	Xus_TN_INPUT_CONTROL.usa_TN_INPUT_CONTROL_DATA[1].by_Attr_mF := BYTE#16#07; (* Weiss, Grün *)
	Xus_TN_INPUT_CONTROL.usa_TN_INPUT_CONTROL_DATA[1].by_Attr_oF := BYTE#16#70; (* Weiss, Blau *)
	Xus_TN_INPUT_CONTROL.usa_TN_INPUT_CONTROL_DATA[1].in_Cursor_Pos := INT#0;
	Xus_TN_INPUT_CONTROL.usa_TN_INPUT_CONTROL_DATA[1].bo_Input_Only_Num := TRUE;
	Xus_TN_INPUT_CONTROL.usa_TN_INPUT_CONTROL_DATA[1].bo_Input_Hidden := FALSE;
	Xus_TN_INPUT_CONTROL.usa_TN_INPUT_CONTROL_DATA[1].st_Input_Mask := '   .   .   .   ';
	Xus_TN_INPUT_CONTROL.usa_TN_INPUT_CONTROL_DATA[1].st_Input_Data := Xus_TN_INPUT_CONTROL.usa_TN_INPUT_CONTROL_DATA[1].st_Input_Mask;
	Xus_TN_INPUT_CONTROL.usa_TN_INPUT_CONTROL_DATA[1].st_Input_ToolTip := 'Enter Agent IP Address in decimal dot format (e.g., 209.131.209.13)';
	Xus_TN_INPUT_CONTROL.usa_TN_INPUT_CONTROL_DATA[1].in_Input_Option := INT#01;
	Xus_TN_INPUT_CONTROL.usa_TN_INPUT_CONTROL_DATA[1].in_Title_Y_Offset := INT#00;
	Xus_TN_INPUT_CONTROL.usa_TN_INPUT_CONTROL_DATA[1].in_Title_X_Offset := -27;
	Xus_TN_INPUT_CONTROL.usa_TN_INPUT_CONTROL_DATA[1].by_Title_Attr := BYTE#16#70;
	Xus_TN_INPUT_CONTROL.usa_TN_INPUT_CONTROL_DATA[1].st_Title_String := 'IP Address              : [149.208.100.100]';

	Xus_TN_INPUT_CONTROL.usa_TN_INPUT_CONTROL_DATA[2].in_Type := INT#01;
	Xus_TN_INPUT_CONTROL.usa_TN_INPUT_CONTROL_DATA[2].in_Y := INT#05;
	Xus_TN_INPUT_CONTROL.usa_TN_INPUT_CONTROL_DATA[2].in_X := INT#44;
	Xus_TN_INPUT_CONTROL.usa_TN_INPUT_CONTROL_DATA[2].by_Attr_mF := BYTE#16#07; (* Weiss, Grün *)
	Xus_TN_INPUT_CONTROL.usa_TN_INPUT_CONTROL_DATA[2].by_Attr_oF := BYTE#16#70; (* Weiss, Blau *)
	Xus_TN_INPUT_CONTROL.usa_TN_INPUT_CONTROL_DATA[2].in_Cursor_Pos := INT#0;
	Xus_TN_INPUT_CONTROL.usa_TN_INPUT_CONTROL_DATA[2].bo_Input_Only_Num := TRUE;
	Xus_TN_INPUT_CONTROL.usa_TN_INPUT_CONTROL_DATA[2].bo_Input_Hidden := FALSE;
	Xus_TN_INPUT_CONTROL.usa_TN_INPUT_CONTROL_DATA[2].st_Input_Mask := '   .   .   .   ';
	Xus_TN_INPUT_CONTROL.usa_TN_INPUT_CONTROL_DATA[2].st_Input_Data := Xus_TN_INPUT_CONTROL.usa_TN_INPUT_CONTROL_DATA[1].st_Input_Mask;
	Xus_TN_INPUT_CONTROL.usa_TN_INPUT_CONTROL_DATA[2].st_Input_ToolTip := 'Enter Agent Netmask (e.g., 255.255.255.0)';
	Xus_TN_INPUT_CONTROL.usa_TN_INPUT_CONTROL_DATA[2].in_Input_Option := INT#01;
	Xus_TN_INPUT_CONTROL.usa_TN_INPUT_CONTROL_DATA[2].in_Title_Y_Offset := INT#00;
	Xus_TN_INPUT_CONTROL.usa_TN_INPUT_CONTROL_DATA[2].in_Title_X_Offset := -27;
	Xus_TN_INPUT_CONTROL.usa_TN_INPUT_CONTROL_DATA[2].by_Title_Attr := BYTE#16#70;
	Xus_TN_INPUT_CONTROL.usa_TN_INPUT_CONTROL_DATA[2].st_Title_String := 'Subnet Mask             : [255.255.255.128]';

	Xus_TN_INPUT_CONTROL.usa_TN_INPUT_CONTROL_DATA[3].in_Type := INT#01;
	Xus_TN_INPUT_CONTROL.usa_TN_INPUT_CONTROL_DATA[3].in_Y := INT#06;
	Xus_TN_INPUT_CONTROL.usa_TN_INPUT_CONTROL_DATA[3].in_X := INT#44;
	Xus_TN_INPUT_CONTROL.usa_TN_INPUT_CONTROL_DATA[3].by_Attr_mF := BYTE#16#07; (* Weiss, Grün *)
	Xus_TN_INPUT_CONTROL.usa_TN_INPUT_CONTROL_DATA[3].by_Attr_oF := BYTE#16#70; (* Weiss, Blau *)
	Xus_TN_INPUT_CONTROL.usa_TN_INPUT_CONTROL_DATA[3].in_Cursor_Pos := INT#0;
	Xus_TN_INPUT_CONTROL.usa_TN_INPUT_CONTROL_DATA[3].bo_Input_Only_Num := TRUE;
	Xus_TN_INPUT_CONTROL.usa_TN_INPUT_CONTROL_DATA[3].bo_Input_Hidden := FALSE;
	Xus_TN_INPUT_CONTROL.usa_TN_INPUT_CONTROL_DATA[3].st_Input_Mask := '   .   .   .   ';
	Xus_TN_INPUT_CONTROL.usa_TN_INPUT_CONTROL_DATA[3].st_Input_Data := Xus_TN_INPUT_CONTROL.usa_TN_INPUT_CONTROL_DATA[1].st_Input_Mask;
	Xus_TN_INPUT_CONTROL.usa_TN_INPUT_CONTROL_DATA[3].st_Input_ToolTip := 'Enter Agent Default Gateway, (e.g., 209.131.209.1)';
	Xus_TN_INPUT_CONTROL.usa_TN_INPUT_CONTROL_DATA[3].in_Input_Option := INT#01;
	Xus_TN_INPUT_CONTROL.usa_TN_INPUT_CONTROL_DATA[3].in_Title_Y_Offset := INT#00;
	Xus_TN_INPUT_CONTROL.usa_TN_INPUT_CONTROL_DATA[3].in_Title_X_Offset := -27;
	Xus_TN_INPUT_CONTROL.usa_TN_INPUT_CONTROL_DATA[3].by_Title_Attr := BYTE#16#70;
	Xus_TN_INPUT_CONTROL.usa_TN_INPUT_CONTROL_DATA[3].st_Title_String := 'Default Gateway         : [149.208.100.1  ]';

	Xus_TN_INPUT_CONTROL.usa_TN_INPUT_CONTROL_DATA[4].in_Type := INT#02;
	Xus_TN_INPUT_CONTROL.usa_TN_INPUT_CONTROL_DATA[4].in_Y := INT#07;
	Xus_TN_INPUT_CONTROL.usa_TN_INPUT_CONTROL_DATA[4].in_X := INT#44;
	Xus_TN_INPUT_CONTROL.usa_TN_INPUT_CONTROL_DATA[4].by_Attr_mF := BYTE#16#07;
	Xus_TN_INPUT_CONTROL.usa_TN_INPUT_CONTROL_DATA[4].by_Attr_oF := BYTE#16#70;
	Xus_TN_INPUT_CONTROL.usa_TN_INPUT_CONTROL_DATA[4].st_Input_Mask := '       ';
	Xus_TN_INPUT_CONTROL.usa_TN_INPUT_CONTROL_DATA[4].st_Input_Data := 'BootP  #DHCP   #DCP    #Static ';
	Xus_TN_INPUT_CONTROL.usa_TN_INPUT_CONTROL_DATA[4].st_Input_ToolTip := 'Push SPACE to select the address assignment (effective after reboot)';
	Xus_TN_INPUT_CONTROL.usa_TN_INPUT_CONTROL_DATA[4].in_Input_Option := INT#02;
	Xus_TN_INPUT_CONTROL.usa_TN_INPUT_CONTROL_DATA[4].in_Title_Y_Offset := INT#00;
	Xus_TN_INPUT_CONTROL.usa_TN_INPUT_CONTROL_DATA[4].in_Title_X_Offset := -27;
	Xus_TN_INPUT_CONTROL.usa_TN_INPUT_CONTROL_DATA[4].by_Title_Attr := BYTE#16#70;
	Xus_TN_INPUT_CONTROL.usa_TN_INPUT_CONTROL_DATA[4].st_Title_String := 'IP Parameter Assignment : <BootP  >';

	Xus_TN_INPUT_CONTROL.usa_TN_INPUT_CONTROL_DATA[5].in_Type := INT#02;
	Xus_TN_INPUT_CONTROL.usa_TN_INPUT_CONTROL_DATA[5].in_Y := INT#09;
	Xus_TN_INPUT_CONTROL.usa_TN_INPUT_CONTROL_DATA[5].in_X := INT#44;
	Xus_TN_INPUT_CONTROL.usa_TN_INPUT_CONTROL_DATA[5].by_Attr_mF := BYTE#16#07;
	Xus_TN_INPUT_CONTROL.usa_TN_INPUT_CONTROL_DATA[5].by_Attr_oF := BYTE#16#70;
	Xus_TN_INPUT_CONTROL.usa_TN_INPUT_CONTROL_DATA[5].st_Input_Mask := '                              ';
	Xus_TN_INPUT_CONTROL.usa_TN_INPUT_CONTROL_DATA[5].st_Input_Data := 'No Redundancy#Rapid Spanning Tree, Disabled#Rapid Spanning Tree, Enabled';
	Xus_TN_INPUT_CONTROL.usa_TN_INPUT_CONTROL_DATA[5].st_Input_ToolTip := 'Push SPACE to chose redundancy (network disruption for few seconds if enabled)';
	Xus_TN_INPUT_CONTROL.usa_TN_INPUT_CONTROL_DATA[5].in_Input_Option := INT#02;
	Xus_TN_INPUT_CONTROL.usa_TN_INPUT_CONTROL_DATA[5].in_Title_Y_Offset := INT#00;
	Xus_TN_INPUT_CONTROL.usa_TN_INPUT_CONTROL_DATA[5].in_Title_X_Offset := -27;
	Xus_TN_INPUT_CONTROL.usa_TN_INPUT_CONTROL_DATA[5].by_Title_Attr := BYTE#16#70;
	Xus_TN_INPUT_CONTROL.usa_TN_INPUT_CONTROL_DATA[5].st_Title_String := 'Redundancy              : <No Redundancy                 >';

	(* Statische Texte ausgeben *)
	FB_TN_SC_WRITE(	Iin_X := INT#17,
					Iin_Y := INT#10,
					Iby_ATTR := BYTE#16#70,
					Ist_STRING := 'Current Vlan Status     :  VLAN Transparent',
					Xus_TN_SCREEN := Xus_TN_SCREEN);

	Xus_TN_INPUT_CONTROL.usa_TN_INPUT_CONTROL_DATA[6].in_Type := INT#02;
	Xus_TN_INPUT_CONTROL.usa_TN_INPUT_CONTROL_DATA[6].in_Y := INT#11;
	Xus_TN_INPUT_CONTROL.usa_TN_INPUT_CONTROL_DATA[6].in_X := INT#44;
	Xus_TN_INPUT_CONTROL.usa_TN_INPUT_CONTROL_DATA[6].by_Attr_mF := BYTE#16#07;
	Xus_TN_INPUT_CONTROL.usa_TN_INPUT_CONTROL_DATA[6].by_Attr_oF := BYTE#16#70;
	Xus_TN_INPUT_CONTROL.usa_TN_INPUT_CONTROL_DATA[6].st_Input_Mask := '                        ';
	Xus_TN_INPUT_CONTROL.usa_TN_INPUT_CONTROL_DATA[6].st_Input_Data := 'VLAN Transparent#VLAN Tagging';
	Xus_TN_INPUT_CONTROL.usa_TN_INPUT_CONTROL_DATA[6].st_Input_ToolTip := 'Push SPACE to toggle the VLAN Mode (effective after reboot)';
	Xus_TN_INPUT_CONTROL.usa_TN_INPUT_CONTROL_DATA[6].in_Input_Option := INT#02;
	Xus_TN_INPUT_CONTROL.usa_TN_INPUT_CONTROL_DATA[6].in_Title_Y_Offset := INT#00;
	Xus_TN_INPUT_CONTROL.usa_TN_INPUT_CONTROL_DATA[6].in_Title_X_Offset := -27;
	Xus_TN_INPUT_CONTROL.usa_TN_INPUT_CONTROL_DATA[6].by_Title_Attr := BYTE#16#70;
	Xus_TN_INPUT_CONTROL.usa_TN_INPUT_CONTROL_DATA[6].st_Title_String := 'Vlan Mode               : <VLAN Transparent        >';

	Xus_TN_INPUT_CONTROL.usa_TN_INPUT_CONTROL_DATA[7].in_Type := INT#02;
	Xus_TN_INPUT_CONTROL.usa_TN_INPUT_CONTROL_DATA[7].in_Y := INT#12;
	Xus_TN_INPUT_CONTROL.usa_TN_INPUT_CONTROL_DATA[7].in_X := INT#44;
	Xus_TN_INPUT_CONTROL.usa_TN_INPUT_CONTROL_DATA[7].by_Attr_mF := BYTE#16#07;
	Xus_TN_INPUT_CONTROL.usa_TN_INPUT_CONTROL_DATA[7].by_Attr_oF := BYTE#16#70;
	Xus_TN_INPUT_CONTROL.usa_TN_INPUT_CONTROL_DATA[7].st_Input_Mask := '       ';
	Xus_TN_INPUT_CONTROL.usa_TN_INPUT_CONTROL_DATA[7].st_Input_Data := 'Disable#Enable';
	Xus_TN_INPUT_CONTROL.usa_TN_INPUT_CONTROL_DATA[7].st_Input_ToolTip := 'Push SPACE to Enable/Disable Port Security';
	Xus_TN_INPUT_CONTROL.usa_TN_INPUT_CONTROL_DATA[7].in_Input_Option := INT#02;
	Xus_TN_INPUT_CONTROL.usa_TN_INPUT_CONTROL_DATA[7].in_Title_Y_Offset := INT#00;
	Xus_TN_INPUT_CONTROL.usa_TN_INPUT_CONTROL_DATA[7].in_Title_X_Offset := -27;
	Xus_TN_INPUT_CONTROL.usa_TN_INPUT_CONTROL_DATA[7].by_Title_Attr := BYTE#16#70;
	Xus_TN_INPUT_CONTROL.usa_TN_INPUT_CONTROL_DATA[7].st_Title_String := 'Port Security           : <Disable>';

	Xus_TN_INPUT_CONTROL.usa_TN_INPUT_CONTROL_DATA[8].in_Type := INT#02;
	Xus_TN_INPUT_CONTROL.usa_TN_INPUT_CONTROL_DATA[8].in_Y := INT#13;
	Xus_TN_INPUT_CONTROL.usa_TN_INPUT_CONTROL_DATA[8].in_X := INT#44;
	Xus_TN_INPUT_CONTROL.usa_TN_INPUT_CONTROL_DATA[8].by_Attr_mF := BYTE#16#07;
	Xus_TN_INPUT_CONTROL.usa_TN_INPUT_CONTROL_DATA[8].by_Attr_oF := BYTE#16#70;
	Xus_TN_INPUT_CONTROL.usa_TN_INPUT_CONTROL_DATA[8].st_Input_Mask := '       ';
	Xus_TN_INPUT_CONTROL.usa_TN_INPUT_CONTROL_DATA[8].st_Input_Data := 'Disable#Enable';
	Xus_TN_INPUT_CONTROL.usa_TN_INPUT_CONTROL_DATA[8].st_Input_ToolTip := 'Push SPACE to Enable/Disable Access Control for the WEB Interface';
	Xus_TN_INPUT_CONTROL.usa_TN_INPUT_CONTROL_DATA[8].in_Input_Option := INT#02;
	Xus_TN_INPUT_CONTROL.usa_TN_INPUT_CONTROL_DATA[8].in_Title_Y_Offset := INT#00;
	Xus_TN_INPUT_CONTROL.usa_TN_INPUT_CONTROL_DATA[8].in_Title_X_Offset := -27;
	Xus_TN_INPUT_CONTROL.usa_TN_INPUT_CONTROL_DATA[8].by_Title_Attr := BYTE#16#70;
	Xus_TN_INPUT_CONTROL.usa_TN_INPUT_CONTROL_DATA[8].st_Title_String := 'Access Control for Web  : <Disable>';

	Xus_TN_INPUT_CONTROL.usa_TN_INPUT_CONTROL_DATA[9].in_Type := INT#02;
	Xus_TN_INPUT_CONTROL.usa_TN_INPUT_CONTROL_DATA[9].in_Y := INT#14;
	Xus_TN_INPUT_CONTROL.usa_TN_INPUT_CONTROL_DATA[9].in_X := INT#44;
	Xus_TN_INPUT_CONTROL.usa_TN_INPUT_CONTROL_DATA[9].by_Attr_mF := BYTE#16#07;
	Xus_TN_INPUT_CONTROL.usa_TN_INPUT_CONTROL_DATA[9].by_Attr_oF := BYTE#16#70;
	Xus_TN_INPUT_CONTROL.usa_TN_INPUT_CONTROL_DATA[9].st_Input_Mask := '        ';
	Xus_TN_INPUT_CONTROL.usa_TN_INPUT_CONTROL_DATA[9].st_Input_Data := 'Default#Profinet';
	Xus_TN_INPUT_CONTROL.usa_TN_INPUT_CONTROL_DATA[9].st_Input_ToolTip := 'Push SPACE to select the switch operating mode';
	Xus_TN_INPUT_CONTROL.usa_TN_INPUT_CONTROL_DATA[9].in_Input_Option := INT#02;
	Xus_TN_INPUT_CONTROL.usa_TN_INPUT_CONTROL_DATA[9].in_Title_Y_Offset := INT#00;
	Xus_TN_INPUT_CONTROL.usa_TN_INPUT_CONTROL_DATA[9].in_Title_X_Offset := -27;
	Xus_TN_INPUT_CONTROL.usa_TN_INPUT_CONTROL_DATA[9].by_Title_Attr := BYTE#16#70;
	Xus_TN_INPUT_CONTROL.usa_TN_INPUT_CONTROL_DATA[9].st_Title_String := 'Switch Operating Mode   : <Default >';

	Xus_TN_INPUT_CONTROL.usa_TN_INPUT_CONTROL_DATA[10].in_Type := INT#02;
	Xus_TN_INPUT_CONTROL.usa_TN_INPUT_CONTROL_DATA[10].in_Y := INT#16;
	Xus_TN_INPUT_CONTROL.usa_TN_INPUT_CONTROL_DATA[10].in_X := INT#44;
	Xus_TN_INPUT_CONTROL.usa_TN_INPUT_CONTROL_DATA[10].by_Attr_mF := BYTE#16#07;
	Xus_TN_INPUT_CONTROL.usa_TN_INPUT_CONTROL_DATA[10].by_Attr_oF := BYTE#16#70;
	Xus_TN_INPUT_CONTROL.usa_TN_INPUT_CONTROL_DATA[10].st_Input_Mask := '       ';
	Xus_TN_INPUT_CONTROL.usa_TN_INPUT_CONTROL_DATA[10].st_Input_Data := 'Enable#Disable';
	Xus_TN_INPUT_CONTROL.usa_TN_INPUT_CONTROL_DATA[10].st_Input_ToolTip := 'Push SPACE to Enable/Disable Web Interface (effective after reboot)';
	Xus_TN_INPUT_CONTROL.usa_TN_INPUT_CONTROL_DATA[10].in_Input_Option := INT#02;
	Xus_TN_INPUT_CONTROL.usa_TN_INPUT_CONTROL_DATA[10].in_Title_Y_Offset := INT#00;
	Xus_TN_INPUT_CONTROL.usa_TN_INPUT_CONTROL_DATA[10].in_Title_X_Offset := -27;
	Xus_TN_INPUT_CONTROL.usa_TN_INPUT_CONTROL_DATA[10].by_Title_Attr := BYTE#16#70;
	Xus_TN_INPUT_CONTROL.usa_TN_INPUT_CONTROL_DATA[10].st_Title_String := 'Web Interface           : <Enable >';

	Xus_TN_INPUT_CONTROL.usa_TN_INPUT_CONTROL_DATA[11].in_Type := INT#02;
	Xus_TN_INPUT_CONTROL.usa_TN_INPUT_CONTROL_DATA[11].in_Y := INT#17;
	Xus_TN_INPUT_CONTROL.usa_TN_INPUT_CONTROL_DATA[11].in_X := INT#44;
	Xus_TN_INPUT_CONTROL.usa_TN_INPUT_CONTROL_DATA[11].by_Attr_mF := BYTE#16#07;
	Xus_TN_INPUT_CONTROL.usa_TN_INPUT_CONTROL_DATA[11].by_Attr_oF := BYTE#16#70;
	Xus_TN_INPUT_CONTROL.usa_TN_INPUT_CONTROL_DATA[11].st_Input_Mask := '       ';
	Xus_TN_INPUT_CONTROL.usa_TN_INPUT_CONTROL_DATA[11].st_Input_Data := 'Enable#Disable';
	Xus_TN_INPUT_CONTROL.usa_TN_INPUT_CONTROL_DATA[11].st_Input_ToolTip := 'Push SPACE to Enable/Disable Telnet Interface (effective after reboot)';
	Xus_TN_INPUT_CONTROL.usa_TN_INPUT_CONTROL_DATA[11].in_Input_Option := INT#02;
	Xus_TN_INPUT_CONTROL.usa_TN_INPUT_CONTROL_DATA[11].in_Title_Y_Offset := INT#00;
	Xus_TN_INPUT_CONTROL.usa_TN_INPUT_CONTROL_DATA[11].in_Title_X_Offset := -27;
	Xus_TN_INPUT_CONTROL.usa_TN_INPUT_CONTROL_DATA[11].by_Title_Attr := BYTE#16#70;
	Xus_TN_INPUT_CONTROL.usa_TN_INPUT_CONTROL_DATA[11].st_Title_String := 'Telnet Interface        : <Enable >';

	Xus_TN_INPUT_CONTROL.usa_TN_INPUT_CONTROL_DATA[12].in_Type := INT#02;
	Xus_TN_INPUT_CONTROL.usa_TN_INPUT_CONTROL_DATA[12].in_Y := INT#18;
	Xus_TN_INPUT_CONTROL.usa_TN_INPUT_CONTROL_DATA[12].in_X := INT#44;
	Xus_TN_INPUT_CONTROL.usa_TN_INPUT_CONTROL_DATA[12].by_Attr_mF := BYTE#16#07;
	Xus_TN_INPUT_CONTROL.usa_TN_INPUT_CONTROL_DATA[12].by_Attr_oF := BYTE#16#70;
	Xus_TN_INPUT_CONTROL.usa_TN_INPUT_CONTROL_DATA[12].st_Input_Mask := '       ';
	Xus_TN_INPUT_CONTROL.usa_TN_INPUT_CONTROL_DATA[12].st_Input_Data := 'Enable#Disable';
	Xus_TN_INPUT_CONTROL.usa_TN_INPUT_CONTROL_DATA[12].st_Input_ToolTip := 'Push SPACE to Enable/Disable SNMP Interface (effective after reboot)';
	Xus_TN_INPUT_CONTROL.usa_TN_INPUT_CONTROL_DATA[12].in_Input_Option := INT#02;
	Xus_TN_INPUT_CONTROL.usa_TN_INPUT_CONTROL_DATA[12].in_Title_Y_Offset := INT#00;
	Xus_TN_INPUT_CONTROL.usa_TN_INPUT_CONTROL_DATA[12].in_Title_X_Offset := -27;
	Xus_TN_INPUT_CONTROL.usa_TN_INPUT_CONTROL_DATA[12].by_Title_Attr := BYTE#16#70;
	Xus_TN_INPUT_CONTROL.usa_TN_INPUT_CONTROL_DATA[12].st_Title_String := 'SNMP Interface          : <Enable >';

	Xus_TN_INPUT_CONTROL.usa_TN_INPUT_CONTROL_DATA[13].in_Type := INT#02;
	Xus_TN_INPUT_CONTROL.usa_TN_INPUT_CONTROL_DATA[13].in_Y := INT#20;
	Xus_TN_INPUT_CONTROL.usa_TN_INPUT_CONTROL_DATA[13].in_X := INT#44;
	Xus_TN_INPUT_CONTROL.usa_TN_INPUT_CONTROL_DATA[13].by_Attr_mF := BYTE#16#07;
	Xus_TN_INPUT_CONTROL.usa_TN_INPUT_CONTROL_DATA[13].by_Attr_oF := BYTE#16#70;
	Xus_TN_INPUT_CONTROL.usa_TN_INPUT_CONTROL_DATA[13].st_Input_Mask := '                                 ';
	Xus_TN_INPUT_CONTROL.usa_TN_INPUT_CONTROL_DATA[13].st_Input_Data := 'No reset#Reset Switch#Reset Switch to factory defaults';
	Xus_TN_INPUT_CONTROL.usa_TN_INPUT_CONTROL_DATA[13].st_Input_ToolTip := 'Push SPACE to select Reset Option';
	Xus_TN_INPUT_CONTROL.usa_TN_INPUT_CONTROL_DATA[13].in_Input_Option := INT#02;
	Xus_TN_INPUT_CONTROL.usa_TN_INPUT_CONTROL_DATA[13].in_Title_Y_Offset := INT#00;
	Xus_TN_INPUT_CONTROL.usa_TN_INPUT_CONTROL_DATA[13].in_Title_X_Offset := -27;
	Xus_TN_INPUT_CONTROL.usa_TN_INPUT_CONTROL_DATA[13].by_Title_Attr := BYTE#16#70;
	Xus_TN_INPUT_CONTROL.usa_TN_INPUT_CONTROL_DATA[13].st_Title_String := 'Reset                   : <No reset                         >';

	Xus_TN_INPUT_CONTROL.usa_TN_INPUT_CONTROL_DATA[14].in_Type := INT#02;
	Xus_TN_INPUT_CONTROL.usa_TN_INPUT_CONTROL_DATA[14].in_Y := INT#22;
	Xus_TN_INPUT_CONTROL.usa_TN_INPUT_CONTROL_DATA[14].in_X := INT#18;
	Xus_TN_INPUT_CONTROL.usa_TN_INPUT_CONTROL_DATA[14].by_Attr_mF := BYTE#16#07;
	Xus_TN_INPUT_CONTROL.usa_TN_INPUT_CONTROL_DATA[14].by_Attr_oF := BYTE#16#70;
	Xus_TN_INPUT_CONTROL.usa_TN_INPUT_CONTROL_DATA[14].st_Input_ToolTip := 'Apply and save ALL changes to permanent memory';
	Xus_TN_INPUT_CONTROL.usa_TN_INPUT_CONTROL_DATA[14].in_Input_Option := INT#01;
	Xus_TN_INPUT_CONTROL.usa_TN_INPUT_CONTROL_DATA[14].in_Title_Y_Offset := INT#00;
	Xus_TN_INPUT_CONTROL.usa_TN_INPUT_CONTROL_DATA[14].in_Title_X_Offset := INT#00;
	Xus_TN_INPUT_CONTROL.usa_TN_INPUT_CONTROL_DATA[14].by_Title_Attr := BYTE#16#70;
	Xus_TN_INPUT_CONTROL.usa_TN_INPUT_CONTROL_DATA[14].st_Title_String := '';
	Xus_TN_INPUT_CONTROL.usa_TN_INPUT_CONTROL_DATA[14].st_Input_Mask := '    ';
	Xus_TN_INPUT_CONTROL.usa_TN_INPUT_CONTROL_DATA[14].st_Input_Data := 'SAVE';

	Xus_TN_INPUT_CONTROL.usa_TN_INPUT_CONTROL_DATA[15].in_Type := INT#02;
	Xus_TN_INPUT_CONTROL.usa_TN_INPUT_CONTROL_DATA[15].in_Y := INT#22;
	Xus_TN_INPUT_CONTROL.usa_TN_INPUT_CONTROL_DATA[15].in_X := INT#11;
	Xus_TN_INPUT_CONTROL.usa_TN_INPUT_CONTROL_DATA[15].by_Attr_mF := BYTE#16#07;
	Xus_TN_INPUT_CONTROL.usa_TN_INPUT_CONTROL_DATA[15].by_Attr_oF := BYTE#16#70;
	Xus_TN_INPUT_CONTROL.usa_TN_INPUT_CONTROL_DATA[15].st_Input_ToolTip := 'Apply changes';
	Xus_TN_INPUT_CONTROL.usa_TN_INPUT_CONTROL_DATA[15].in_Input_Option := INT#01;
	Xus_TN_INPUT_CONTROL.usa_TN_INPUT_CONTROL_DATA[15].in_Title_Y_Offset := INT#00;
	Xus_TN_INPUT_CONTROL.usa_TN_INPUT_CONTROL_DATA[15].in_Title_X_Offset := INT#00;
	Xus_TN_INPUT_CONTROL.usa_TN_INPUT_CONTROL_DATA[15].by_Title_Attr := BYTE#16#70;
	Xus_TN_INPUT_CONTROL.usa_TN_INPUT_CONTROL_DATA[15].st_Title_String := '';
	Xus_TN_INPUT_CONTROL.usa_TN_INPUT_CONTROL_DATA[15].st_Input_Mask := '     ';
	Xus_TN_INPUT_CONTROL.usa_TN_INPUT_CONTROL_DATA[15].st_Input_Data := 'APPLY';

	Xus_TN_INPUT_CONTROL.usa_TN_INPUT_CONTROL_DATA[16].in_Type := INT#02;
	Xus_TN_INPUT_CONTROL.usa_TN_INPUT_CONTROL_DATA[16].in_Y := INT#22;
	Xus_TN_INPUT_CONTROL.usa_TN_INPUT_CONTROL_DATA[16].in_X := INT#03;
	Xus_TN_INPUT_CONTROL.usa_TN_INPUT_CONTROL_DATA[16].by_Attr_mF := BYTE#16#07;
	Xus_TN_INPUT_CONTROL.usa_TN_INPUT_CONTROL_DATA[16].by_Attr_oF := BYTE#16#70;
	Xus_TN_INPUT_CONTROL.usa_TN_INPUT_CONTROL_DATA[16].st_Input_ToolTip := 'Return to Main Menu';
	Xus_TN_INPUT_CONTROL.usa_TN_INPUT_CONTROL_DATA[16].in_Input_Option := INT#01;
	Xus_TN_INPUT_CONTROL.usa_TN_INPUT_CONTROL_DATA[16].in_Title_Y_Offset := INT#00;
	Xus_TN_INPUT_CONTROL.usa_TN_INPUT_CONTROL_DATA[16].in_Title_X_Offset := INT#00;
	Xus_TN_INPUT_CONTROL.usa_TN_INPUT_CONTROL_DATA[16].by_Title_Attr := BYTE#16#70;
	Xus_TN_INPUT_CONTROL.usa_TN_INPUT_CONTROL_DATA[16].st_Title_String := '';
	Xus_TN_INPUT_CONTROL.usa_TN_INPUT_CONTROL_DATA[16].st_Input_Mask := '      ';
	Xus_TN_INPUT_CONTROL.usa_TN_INPUT_CONTROL_DATA[16].st_Input_Data := 'LOGOUT';

	(* Control-Tool-Tip *)
	Xus_TN_INPUT_CONTROL.in_ToolTip_Y := INT#23;
	Xus_TN_INPUT_CONTROL.in_ToolTip_X := INT#00;
	Xus_TN_INPUT_CONTROL.by_ToolTip_Attr := BYTE#07;
	Xus_TN_INPUT_CONTROL.in_ToolTip_Size := INT#80;

	(* Control-Verwaltung initialisieren *)
	Xus_TN_INPUT_CONTROL.in_Count := INT#16;
	Xus_TN_INPUT_CONTROL.bo_Enable := TRUE;
	Xus_TN_INPUT_CONTROL.bo_Reset_Fokus := TRUE;

END_IF;

IF (Xus_TN_SCREEN.in_Page_Number = INT#05) THEN

	(* eingegebenen String übernehmen *)
	IF Xus_TN_INPUT_CONTROL.usa_TN_INPUT_CONTROL_DATA[16].bo_Input_Entered = TRUE THEN

		Xus_TN_INPUT_CONTROL.usa_TN_INPUT_CONTROL_DATA[16].bo_Input_Entered := FALSE;
		Xus_TN_SCREEN.in_Page_Number := INT#00;
	END_IF;
END_IF;

END_PROGRAM

// ---- POUs/DEMO/WORLD_WEATHER_DEMO.TcPOU
PROGRAM WORLD_WEATHER_DEMO
VAR
	IP_C: IP_C;
	S_BUF: NETWORK_BUFFER;
	R_BUF: NETWORK_BUFFER;
	IP_CONTROL_1: IP_CONTROL;
	activate: BOOL := TRUE;
	done: BOOL;
	busy: BOOL;
	error_c: DWORD;
	error_t: BYTE;
	latitude: REAL := 48.21;
	longitude: REAL := 16.37;
	WORLD_WEATHER: WORLD_WEATHER;
	WW_DATA: WORLD_WEATHER_DATA;
	CLK_PRG: CLK_PRG;
	WORLD_WEATHER_DESC_GE: WORLD_WEATHER_DESC_GE;
	WORLD_WEATHER_ICON_OSCAT: WORLD_WEATHER_ICON_OSCAT;
END_VAR
VAR // added by the converter: edge detectors and wires of the graphical bodies
    _w1 : ANY;
END_VAR

CLK_PRG(_in1 := t#3h);
activate := CLK_PRG._out1;
WORLD_WEATHER(
    ACTIVATE := activate,
    LATITUDE := latitude,
    LONGITUDE := longitude,
    KEY := '5c6ecef5cc131759100310',
    IP_C := IP_C,
    S_BUF := S_BUF,
    R_BUF := R_BUF,
    WW := WW_DATA);
busy := WORLD_WEATHER.BUSY;
done := WORLD_WEATHER.DONE;
error_c := WORLD_WEATHER.ERROR_C;
error_t := WORLD_WEATHER.ERROR_T;
// Wetterbeschreibung auf Deutsch (optional)
WORLD_WEATHER_DESC_GE(ACTIVATE := done, WW := WW_DATA);
// ICONS nach OSCAT-Standard (optional)
WORLD_WEATHER_ICON_OSCAT(ACTIVATE := done, WW := WW_DATA);
// IP-Adresse des DNS-Server oder des DSL-Router
_w1 := DWORD_OF_BYTE(8, 8, 8, 8);
IP_CONTROL_1(IP := _w1, TIME_OUT := T#5s, IP_C := IP_C, S_BUF := S_BUF, R_BUF := R_BUF); // IP_CONTROL

END_PROGRAM

// ---- POUs/WEATHER/WORLD_WEATHER.TcPOU
FUNCTION_BLOCK WORLD_WEATHER
VAR_IN_OUT
	IP_C : IP_C; (* IP_Control Verwaltungsstruktur *)
	S_BUF : NETWORK_BUFFER;
	R_BUF : NETWORK_BUFFER;
	WW : WORLD_WEATHER_DATA;
END_VAR
VAR_INPUT
	ACTIVATE : BOOL;
	LATITUDE : REAL;
	LONGITUDE : REAL;
	KEY : STRING(30);
END_VAR
VAR_OUTPUT
	BUSY : BOOL;
	DONE : BOOL;
	ERROR_C : DWORD;
	ERROR_T : BYTE;
END_VAR
VAR
	URL_DATA : url;
	DNS_CLIENT : DNS_CLIENT;
	HTTP_GET : HTTP_GET;
	CPB : CSV_PARSER_BUF;
	last_state : BOOL;
	value_int : INT;
	value_real : REAL;
	v_real : REAL;
	state : INT;
	url_str : T_MaxString;
	offset : UDINT;
	size : INT;
	sep : BYTE;
	cnt : INT;
	day : INT;
	idx : INT;
	run : BYTE;
	result : BYTE;
	value : T_MaxString;
	pos : INT;
END_VAR

(*

version 1.3	05. jan 2012
programmer 	ks
tested by		ks

WORLD_WEATHER lädt von worldweather.com eine Wetter csv-datei und analysiert die Daten und legt diese in einem Array ab
Die Wetterdaten werden für 5 tage aufbereitet

*)

CASE state OF

00:
	IF ACTIVATE AND NOT last_state THEN
		state := 20;
		DONE := FALSE;
		BUSY := TRUE;
		ERROR_C := DWORD#0;
		ERROR_T := BYTE#0;
	END_IF;

20: (* URL for DNS UND HTTP-GET *)
	(* Example: http://free.worldweatheronline.com/feed/weather.ashx?q=48.21,16.37&format=csv&num_of_days=5&key=xxxxxxxxxxxxxxxxxxxxxx *)
	url_str := CONCAT('http://free.worldweatheronline.com/feed/weather.ashx?q=',REAL_TO_STRF(LATITUDE,6,D:='.'));
	url_str := CONCAT(url_str,',');
	url_str := CONCAT(url_str,REAL_TO_STRF(LONGITUDE,6,D:='.'));
	url_str := CONCAT(url_str,'&format=csv&num_of_days=5&key=');
	url_str := CONCAT(url_str,key);

	URL_DATA:=STRING_TO_URL(STR:=url_str, DEFAULT_PROTOCOL:='', DEFAULT_PATH:='' );
	state := 40;

40:
	IF DNS_CLIENT.DONE THEN
		state := 60;
	ELSIF (DNS_CLIENT.ERROR > DWORD#00) THEN
		(* Fehlerbehandlung *)
		ERROR_C := DNS_CLIENT.ERROR;
	ERROR_T := BYTE#01;
		state   := 100;
	END_IF;

60:
	IF HTTP_GET.DONE THEN
		sep := 0;
		idx := 0;
		day := 0;
		cnt := 0;
		OFFSET := HTTP_GET.BODY_START; (* Start Offset vorgeben *)
		size := HTTP_GET.BODY_STOP; (* End Position *)
		run := 1; (* Element suchen *)
		state := 80;

	ELSIF (HTTP_GET.ERROR > DWORD#00) THEN
		(* Fehlerbehandlung *)
		ERROR_C := HTTP_GET.ERROR;
		ERROR_T := BYTE#02;
		state := 100;
	END_IF;

80:	IF run = 0 THEN (* kein Befehl mehr aktiv ? *)
		run := 1; (*  nächstes Element suchen  *)
		IF result = 1 OR result = 2 THEN
			value_int := 0;
			value_real := 0.0;
			(* automatische konvertierung in real und int ausführen *)
			IF LEN(value) <= 20 THEN
				v_real:=FLOAT_TO_REAL(FLT:=value);
				IF CHK_REAL(v_real) = 0 THEN (* !!! prüft auf gültigen REAL Wert, ansonsten stürzt Twincat ab !!!!  *)
					value_real := v_real;
					value_int := REAL_TO_INT(value_real);
				END_IF;
			END_IF;
			cnt := cnt + 1;
			IF cnt >=8 AND cnt <= 87 THEN
				IF cnt > 22 THEN
					CASE idx OF
					00:	WW.DAY[day].DATE_OF_DAY := value;
					01:	WW.DAY[day].TEMP_MAX_C := value_int;
					02:	WW.DAY[day].TEMP_MAX_F := value_int;
					03:	WW.DAY[day].TEMP_MIN_C := value_int;
					04:	WW.DAY[day].TEMP_MIN_F := value_int;
					05:	WW.DAY[day].WIND_SPEED_MILES := value_int;
					06:	WW.DAY[day].WIND_SPEED_KMPH := value_int;
					07:	WW.DAY[day].WIND_DIR_DEGREE := value_int;
					08:	WW.DAY[day].WIND_DIR16POINT := value;
					09:	WW.DAY[day].WEATHER_CODE := value_int;
					10:	pos := FIND(value, '/wsymbol_');
						WW.DAY[day].WEATHER_ICON := DEC_TO_INT(MID(value,4,pos+9));
					11:	WW.DAY[day].WEATHER_DESC := value;
					12:	WW.DAY[day].PRECIPMM := value_real;
					END_CASE;
					idx := idx + 1;
					IF idx > 12 THEN
						idx := 0;
						day := day + 1;
					END_IF;
				ELSE
					CASE cnt OF
					08:	sep :=44; (* ab jetzt mit Trennzeichen arbeiten, *)
					09:	WW.CUR.OBSERVATION_TIME := value;
					10:	WW.CUR.TEMP_C := value_int;
					11:	WW.CUR.WEATHER_CODE := value_int;
					12:	pos := FIND(value, '/wsymbol_');
						WW.CUR.WEATHER_ICON := DEC_TO_INT(MID(value,4,pos+9));
					13:	WW.CUR.WEATHER_DESC := value;
					14:	WW.CUR.WIND_SPEED_MILES := value_int;
					15:	WW.CUR.WIND_SPEED_KMPH := value_int;
					16:	WW.CUR.WIND_DIR_DEGREE := value_int;
					17:	WW.CUR.WIND_DIR16POINT := value;
					18:	WW.CUR.PRECIPMM := value_real;
					19:	WW.CUR.HUMIDITY := value_int;
					20:	WW.CUR.VISIBILITY := value_int;
					21:	WW.CUR.PRESSURE := value_int;
					22:	WW.CUR.CLOUDOVER := value_int;
					END_CASE;
				END_IF;
			END_IF;
		ELSIF result = 10 THEN (* nichts mehr gefunden *)
			DONE  := TRUE;
			run := 0; (* Auswertung beenden *)
			state := 100;
		END_IF;
	END_IF;

100:
	(* UNLOCK HTTP DATA *)
	IF (NOT HTTP_GET.DONE) THEN
		state := 0;
		BUSY := FALSE;
		DONE := ERROR_T = BYTE#0;
	END_IF;

END_CASE;

(* ---------------- DNS --------------- *)
DNS_CLIENT(	IP_C:=IP_C,
			S_BUF:=S_BUF,
			R_BUF:=R_BUF,
			DOMAIN:=URL_DATA.DOMAIN,
			IP4_DNS:=DWORD#00,
			ACTIVATE:=state=40 (* DNS Start *)
			);
(* nicht oder nicht direkt verwendete Parameter *)
(*	DWORD :=DNS_CLIENT.IP4;
	BOOL  :=DNS_CLIENT.DONE;
	BYTE  :=DNS_CLIENT.ERROR; *)
(* -------------------------------------*)

(* ------------- HTTP_GET --------------- *)
HTTP_GET(	IP_C:=IP_C,
			S_BUF:=S_BUF,
			R_BUF:=R_BUF,
			IP4:=DNS_CLIENT.IP4,
			GET:=state=60,
			MODE:=BYTE#2, (* HTTP 1.1 mit persistenter Verbindung *)
			UNLOCK_BUF:=state=100,
			URL_DATA:=URL_DATA
			);

(* nicht oder nicht direkt verwendete Parameter *)
(*	STRING := HTTP_GET.HTTP_STATUS;
	UINT :=HTTP_GET.HEADER_START;
	UINT :=HTTP_GET.HEADER_STOP;
	UINT :=HTTP_GET.BODY_START;
	UINT :=HTTP_GET.BODY_STOP;
	BOOL :=HTTP_GET.DONE;
	BYTE :=HTTP_GET.ERROR;
*)
(* -------------------------------------*)
CPB(SEP:=sep,RUN:=run,OFFSET:=OFFSET,VALUE:=value,PT:=R_BUF,RESULT=>result); (* CSV PARAMETER BUF *)

last_state := ACTIVATE;

(* revision history
ks	01.oct. 2010	rev 1.0
	original version

ks	01.feb. 2011	rev 1.1
	rücksetzen von cnt 

ks	07.apr. 2011	rev 1.2
	neue Domain "free.worldweatheronline.com" (Ab 30.04.2011 notwendig)

ks	05.jan. 2012	rev 1.3
	neues datenelement "icon" integriert, REAL_TO_STRF parameter D
*)

END_FUNCTION_BLOCK

// ---- POUs/WEATHER/WORLD_WEATHER_DESC_GE.TcPOU
FUNCTION_BLOCK WORLD_WEATHER_DESC_GE
VAR_IN_OUT
	WW : WORLD_WEATHER_DATA;
END_VAR
VAR_INPUT
	ACTIVATE : BOOL;
END_VAR
VAR
	act_last : BOOL;
	x : INT;
	y : INT;
	str : STRING(60);
	i : INT;
END_VAR

(*

version 1.0		04. may. 2011
programmer 		ks
tested by			ks

WORLD_WEATHER_DESC_GE ändert die englischen Wetterbeschreibungstexte auf deutsche Texte um
*)

IF ACTIVATE AND act_last = FALSE THEN
	i := 0;
	FOR y := 1 TO 12 DO
		CASE y OF
		1,3,5,7,9:		x :=  WW.DAY[i].WEATHER_CODE;
		2,4,6,8,10:	WW.DAY[i].WEATHER_DESC := str;
					i := i + 1;
		11:			x :=  WW.CUR.WEATHER_CODE;
		12:			WW.CUR.WEATHER_DESC := str;
		END_CASE;

		CASE x OF
			113	:	str := 'heiter/sonnig';
			116	:	str := 'stellenweise wolkig';
			119	:	str := 'wolkig';
			122	:	str := 'bewölkt';
			143	:	str := 'Nebel';
			176	:	str := 'stellenweise nahegelegener Regen';
			179	:	str := 'stellenweise nahegelegener Schneefall';
			182	:	str := 'stellenweise nahegelegener Eisregen';
			185	:	str := 'stellenweise gefrierender Niesel';
			200	:	str := 'nahegelegene Sturm';
			227	:	str := 'Schneetreiben';
			230	:	str := 'Schneesturm';
			248	:	str := 'Nebel';
			260	:	str := 'gefrierender Nebel';
			263	:	str := 'stellenweise leichter Nieselregen';
			266	:	str := 'leichter Niesel';
			281	:	str := 'gefrierender Nieselregen';
			284	:	str := 'stark gefrierender Nieselregen';
			293	:	str := 'stellenweise leichter Regen';
			296	:	str := 'leichter Regen';
			299	:	str := 'zeitweise etwas Regen';
			302	:	str := 'mäßiger Regen';
			305	:	str := 'zeitweise etwas starker Regen';
			308	:	str := 'starker Regen';
			311	:	str := 'leichter gefrierender Regen';
			314	:	str := 'mäßiger oder starker Eisregen';
			317	:	str := 'leichter Eisregen';
			320	:	str := 'mäßiger oder starker Eisregen';
			323	:	str := 'stellenweise leichter Schneefall';
			326	:	str := 'leichter Scheefall';
			329	:	str := 'stellenweise moderater Schneefall';
			332	:	str := 'mäßiger Schnee';
			335	:	str := 'stellenweise starker Scheefall';
			338	:	str := 'starker Schneefall';
			350	:	str := 'Hagel';
			353	:	str := 'leichte Regenfälle';
			356	:	str := 'mäßiger oder starker Regenfall';
			359	:	str := 'sintflutartige Regenfälle';
			362	:	str := 'leichter Eisregen';
			365	:	str := 'mäßiger oder starker Eisregen';
			368	:	str := 'leichte Schneeschauer';
			371	:	str := 'mäßiger oder starker Schneefall';
			374	:	str := 'leichter Hagel';
			377	:	str := 'mäßiger oder starker Hagel';
			386	:	str := 'stellenweise leichter Regen in Gewittergebiet';
			389	:	str := 'mäßiger oder starker Regen in Gewittergebiet';
			392	:	str := 'stellenweise leichter Schneefall in Gewittergebiet';
			395	:	str := 'mäßiger oder starker Schnee in Gewittergebiet';
		ELSE
			str := 	'nicht verfügbar';
		END_CASE;
	END_FOR;
END_IF;
act_last := ACTIVATE;

(* revision history
ks	04. may. 2011	rev 1.0
	original version
*)

END_FUNCTION_BLOCK

// ---- POUs/WEATHER/WORLD_WEATHER_ICON_OSCAT.TcPOU
FUNCTION_BLOCK WORLD_WEATHER_ICON_OSCAT
VAR_IN_OUT
	WW : WORLD_WEATHER_DATA;
END_VAR
VAR_INPUT
	ACTIVATE : BOOL;
END_VAR
VAR
	dat : ARRAY[0..41] OF INT := [0,14,12,9,9,0,7,7,0,2,2,3,3,1,0,0,17,4,4,3,3,1,0,0,17,2,2,3,3,1,0,0,17,2,4,3,3,1,0,0,17,0];
	act_last : BOOL;
	x : INT;
	i : INT;
END_VAR

(*

version 1.0		04. may. 2011
programmer 		ks
tested by			ks

WORLD_WEATHER_ICON_OSCAT ändert die ICON Nummer auf den OSCAT-Standard um
*)

IF ACTIVATE AND act_last = FALSE THEN
	x := LIMIT(0,WW.CUR.WEATHER_ICON,41);
	WW.CUR.WEATHER_ICON := dat[x];
	FOR i := 0 TO 4 DO
		x := LIMIT(0,WW.DAY[i].WEATHER_ICON,41);
		WW.DAY[i].WEATHER_ICON := dat[x];
	END_FOR;
END_IF;
act_last := ACTIVATE;

(* revision history
ks	04. may. 2011	rev 1.0
	original version
*)

END_FUNCTION_BLOCK

// ---- POUs/DEMO/YAHOO_WEATHER_DEMO.TcPOU
PROGRAM YAHOO_WEATHER_DEMO
VAR
	IP_C: IP_C;
	S_BUF: NETWORK_BUFFER;
	R_BUF: NETWORK_BUFFER;
	IP_CONTROL_1: IP_CONTROL;
	activate: BOOL;
	done: BOOL;
	busy: BOOL;
	error_c: DWORD;
	error_t: BYTE;
	YAHOO_WEATHER: YAHOO_WEATHER;
	YW_DATA: YAHOO_WEATHER_DATA;
	CLK_PRG: CLK_PRG;
	YAHOO_WEATHER_DESC_GE: YAHOO_WEATHER_DESC_GE;
	YAHOO_WEATHER_ICON_OSCAT: YAHOO_WEATHER_ICON_OSCAT;
END_VAR
VAR // added by the converter: edge detectors and wires of the graphical bodies
    _w1 : ANY;
END_VAR

CLK_PRG(_in1 := t#3h);
activate := CLK_PRG._out1;
YAHOO_WEATHER(
    ACTIVATE := activate,
    UNITS := FALSE,
    LOCATION := '551801',
    IP_C := IP_C,
    S_BUF := S_BUF,
    R_BUF := R_BUF,
    YW := YW_DATA);
busy := YAHOO_WEATHER.BUSY;
done := YAHOO_WEATHER.DONE;
error_c := YAHOO_WEATHER.ERROR_C;
error_t := YAHOO_WEATHER.ERROR_T;
// Wetterbeschreibung auf Deutsch (optional)
YAHOO_WEATHER_DESC_GE(ACTIVATE := done, YW := YW_DATA);
// ICONS nach OSCAT-Standard (optional)
YAHOO_WEATHER_ICON_OSCAT(ACTIVATE := done, YW := YW_DATA);
// IP-Adresse des DNS-Server oder des DSL-Router
_w1 := DWORD_OF_BYTE(8, 8, 8, 8);
IP_CONTROL_1(IP := _w1, TIME_OUT := T#5s, IP_C := IP_C, S_BUF := S_BUF, R_BUF := R_BUF); // IP_CONTROL

END_PROGRAM

// ---- POUs/WEATHER/YAHOO_WEATHER.TcPOU
FUNCTION_BLOCK YAHOO_WEATHER
VAR_IN_OUT
	IP_C : IP_C; (* IP_Control Verwaltungsstruktur *)
	S_BUF : NETWORK_BUFFER;
	R_BUF : NETWORK_BUFFER;
	YW : YAHOO_WEATHER_DATA;
END_VAR
VAR_INPUT
	ACTIVATE : BOOL;
	UNITS : BOOL;
	LOCATION : STRING(20);
END_VAR
VAR_OUTPUT
	BUSY : BOOL;
	DONE : BOOL;
	ERROR_C : DWORD;
	ERROR_T : BYTE;
END_VAR
VAR
	CTRL : XML_CONTROL;
	XML_READER : XML_READER;
	URL_DATA : url;
	DNS_CLIENT : DNS_CLIENT;
	HTTP_GET : HTTP_GET;
	last_state : BOOL;
	value_int : INT;
	value_real : REAL;
	v_real : REAL;
	state : INT;
END_VAR

(*

version 1.3		04. may. 2011
programmer 		ks
tested by			ks

YAHOO_WEATHER lädt vom Yahoo-Webserver einen Wetter RSS-Feed und analysiert die Daten und legt diese in einem Array ab
*)

CASE state OF

00:	IF ACTIVATE AND NOT last_state THEN
		state := 20;
		DONE := FALSE;
		BUSY := TRUE;
		ERROR_C := DWORD#0;
		ERROR_T := BYTE#0;
	END_IF;

20: (* URL for DNS UND HTTP-GET *)
	(* Example: http://weather.yahooapis.com/forecastrss?p=94089&u=c *)
	URL_DATA:=STRING_TO_URL(STR:='http://weather.yahooapis.com/forecastrss',
							DEFAULT_PROTOCOL:='',
							DEFAULT_PATH:=''
							);
  	URL_DATA.QUERY := CONCAT('w=',LOCATION);

	IF UNITS THEN
		URL_DATA.QUERY := CONCAT(URL_DATA.QUERY,'&u=f'); (* fahrenheit *)
	ELSE
		URL_DATA.QUERY := CONCAT(URL_DATA.QUERY,'&u=c'); (* celsius *)
	END_IF;
	state := 40;

40:	IF DNS_CLIENT.DONE THEN
		state := 60;
	ELSIF (DNS_CLIENT.ERROR > DWORD#00) THEN
		(* Fehlerbehandlung *)
		ERROR_C := DNS_CLIENT.ERROR;
	ERROR_T := BYTE#01;
		state   := 100;
	END_IF;

60:	IF HTTP_GET.DONE THEN
		state := 80;
		CTRL.START_POS := HTTP_GET.BODY_START;
		CTRL.STOP_POS := HTTP_GET.BODY_STOP;
		CTRL.COMMAND := WORD#2#10000000_00011000; (* ONLY TEXT AND ATTRIBUTE *)
		CTRL.WATCHDOG  := T#1ms;

	ELSIF (HTTP_GET.ERROR > DWORD#00) THEN
		(* Fehlerbehandlung *)
		ERROR_C := HTTP_GET.ERROR;
		ERROR_T := BYTE#02;
		state := 100;
	END_IF;

80: XML_READER(CTRL:=CTRL,BUF:=R_BUF.BUFFER); (* XML Daten seriell lesen *)
	IF CTRL.TYP < 98 THEN (* nur auswerten wenn kein Watchdog durchlauf *)
		value_int := 0;
		value_real := 0.0;
		(* automatische konvertierung in real und int ausführen *)
		IF LEN(CTRL.VALUE) <= 20 THEN
			v_real:=FLOAT_TO_REAL(FLT:=CTRL.VALUE);
			IF CHK_REAL(v_real) = 0 THEN (* !!! prüft auf gültigen REAL Wert, ansonsten stürzt Twincat ab !!!!  *)
				value_real := v_real;
				value_int := REAL_TO_INT(value_real);
			END_IF;
		END_IF;

		IF CTRL.COUNT < UINT#52 THEN (* Performance-Teilung *)
			(* ------------ Teil 1 --------------*)
			CASE UINT_TO_INT(CTRL.COUNT) OF
			027: YW.TimeToLive := value_int;
			030: YW.location_city := CTRL.VALUE;
			031: YW.location_region := CTRL.VALUE;
			032: YW.location_country := CTRL.VALUE;
			035: YW.unit_temperature := CTRL.VALUE;
			036: YW.unit_distance := CTRL.VALUE;
			037: YW.unit_pressure := CTRL.VALUE;
			038: YW.unit_speed := CTRL.VALUE;
			041: YW.wind_chill := value_int;
			042: YW.wind_direction := value_int;
			043: YW.wind_speed := value_real;
			046: YW.atmosphere_humidity := value_int;
			047: YW.atmosphere_visibility := value_real;
			048: YW.atmosphere_pressure := value_int;
			049: YW.atmosphere_rising := value_int;
			END_CASE;
		ELSE
			(* ------------ Teil 2 --------------*)
			CASE UINT_TO_INT(CTRL.COUNT) OF
			052: YW.astronomy_sunrise := CTRL.VALUE;
			053: YW.astronomy_sunset := CTRL.VALUE;
			077: YW.geo_latitude := value_real;
			080: YW.geo_longitude := value_real;
			089: YW.cur_conditions_text := CTRL.VALUE;
			090: YW.cur_conditions_code := value_int;
				YW.cur_conditions_icon := value_int;
			091: YW.cur_conditions_temp := value_int;
			100: YW.forcast_today_low_temp := value_int;
			101: YW.forcast_today_high_temp := value_int;
			102: YW.forcast_today_text := CTRL.VALUE;
			103: YW.forcast_today_code := value_int;
				YW.forcast_today_icon := value_int;
			108: YW.forcast_tomorrow_low_temp := value_int;
			109: YW.forcast_tomorrow_high_temp := value_int;
			110: YW.forcast_tomorrow_text := CTRL.VALUE;
			111: YW.forcast_tomorrow_code := value_int;
				YW.forcast_tomorrow_icon := value_int;
			END_CASE;
		END_IF;
	ELSIF CTRL.TYP = 99 THEN (* EXIT - letztes Element gelesen *)
		DONE  := TRUE;
		state := 100;
	END_IF; 

100:
	(* UNLOCK HTTP DATA *)
	IF (NOT HTTP_GET.DONE) THEN
		state := 0;
		BUSY := FALSE;
		DONE := ERROR_T = BYTE#0;
	END_IF; 

	END_CASE;

(* ---------------- DNS --------------- *)
DNS_CLIENT(	IP_C:=IP_C,
			S_BUF:=S_BUF,
			R_BUF:=R_BUF,
			DOMAIN:=URL_DATA.DOMAIN,
			IP4_DNS:=DWORD#00,
			ACTIVATE:=state=40 (* DNS Start *)
			);
(* nicht oder nicht direkt verwendete Parameter *)
(*	DWORD :=DNS_CLIENT.IP4;
	BOOL  :=DNS_CLIENT.DONE;
	BYTE  :=DNS_CLIENT.ERROR; *)
(* -------------------------------------*)

(* ------------- HTTP_GET --------------- *)
HTTP_GET(	IP_C:=IP_C,
			S_BUF:=S_BUF,
			R_BUF:=R_BUF,
			IP4:=DNS_CLIENT.IP4,
			GET:=state=60,
			MODE:=BYTE#2, (* HTTP 1.1 mit persistenter Verbindung *)
			UNLOCK_BUF:=state=100,
			URL_DATA:=URL_DATA
			);

(* nicht oder nicht direkt verwendete Parameter *)
(*	STRING := HTTP_GET.HTTP_STATUS;
	UINT :=HTTP_GET.HEADER_START;
	UINT :=HTTP_GET.HEADER_STOP;
	UINT :=HTTP_GET.BODY_START;
	UINT :=HTTP_GET.BODY_STOP;
	BOOL :=HTTP_GET.DONE;
	BYTE :=HTTP_GET.ERROR;
*)
(* -------------------------------------*)

last_state := ACTIVATE;

(* revision history
ks	18. dez. 2008	rev 1.0
	original version

ks	01. oct. 2009	rev 1.1
	YAHOO_WEATHER_DATA

ks	24. sep. 2010	rev 1.2
	new URL-Location-parameter and REAL_CHECK (TwinCat BUG) 

ks	04. may. 2011	rev 1.3
	neue elemente:  CUR_CONDITIONS_ICON, FORCAST_TODAY_ICON, FORCAST_TOMORROW_ICON

*)

END_FUNCTION_BLOCK

// ---- POUs/WEATHER/YAHOO_WEATHER_DESC_GE.TcPOU
FUNCTION_BLOCK YAHOO_WEATHER_DESC_GE
VAR_IN_OUT
	YW : YAHOO_WEATHER_DATA;
END_VAR
VAR_INPUT
	ACTIVATE : BOOL;
END_VAR
VAR
	act_last : BOOL;
	x : INT;
	y : INT;
	str : STRING(40);
END_VAR

(*

version 1.0		04. may. 2011
programmer 		ks
tested by			ks

YAHOO_WEATHER_DESC_GE ändert die englischen Wetterbeschreibungstexte auf deutsche Texte um
*)

IF ACTIVATE AND act_last = FALSE THEN
	FOR y := 1 TO 4 DO
		CASE y OF
		1:	x := YW.CUR_CONDITIONS_CODE;
		2 :	YW.CUR_CONDITIONS_TEXT := str;
			x := YW.FORCAST_TODAY_CODE;
		3 :	YW.FORCAST_TODAY_TEXT := str;
			x := YW.FORCAST_TOMORROW_CODE;
		4 :	YW.FORCAST_TOMORROW_TEXT := str;
		END_CASE;

		CASE x OF
		00:	str := 'Wirbelsturm';
		01:	str := 'Tropensturm';
		02:	str := 'Wirbelsturm';
		03:	str := 'starkes Gewitter ';
		04:	str := 'Gewitter';
		05:	str := 'Schneeregen';
		06:	str := 'Schneeregen';
		07:	str := 'Schneeregen';
		08:	str := 'gefrierender Nieselregen';
		09:	str := 'Nieselregen';
		10:	str := 'gefrierender Regen';
		11:	str := 'Regenfälle';
		12:	str := 'Regenfälle';
		13:	str := 'Schneegestöber';
		14:	str := 'leichte Schneefälle';
		15:	str := 'Schneetreiben';
		16:	str := 'Schnee';
		17:	str := 'Hagel';
		18:	str := 'Schneeregen';
		19:	str := 'Staub';
		20:	str := 'nebelig';
		21:	str := 'Dunst';
		22:	str := 'rauchig';
		23:	str := 'stürmisch';
		24:	str := 'windig';
		25:	str := 'kalt';
		26:	str := 'bewölkt';
		27:	str := 'meist bewölkt';
		28:	str := 'meist bewölkt';
		29:	str := 'teilweise bewölkt';
		30:	str := 'teilweise bewölkt';
		31:	str := 'klar';
		32:	str := 'sonnig';
		33:	str := 'heiter';
		34:	str := 'heiter';
		35:	str := 'Regen und Hagel';
		36:	str := 'heiß';
		37:	str := 'örtliche Gewitter';
		38:	str := 'vereinzelte Gewitter';
		39:	str := 'vereinzelte Gewitter';
		40:	str := 'vereinzelte Regenfälle';
		41:	str := 'schwere Schneefälle';
		42:	str := 'vereinzelte Schneefälle';
		43:	str := 'schwere Schneefälle';
		44:	str := 'teilweise bewölkt';
		45:	str := 'gewittrige Regenfälle';
		46:	str := 'Schneefälle';
		47:	str := 'örtliche gewittrige Regenfälle';
		ELSE
			str := 'nicht verfügbar';
		END_CASE;
	END_FOR;
END_IF;
act_last := ACTIVATE;

(* revision history
ks	04. may. 2011	rev 1.0
	original version
*)

END_FUNCTION_BLOCK

// ---- POUs/WEATHER/YAHOO_WEATHER_ICON_OSCAT.TcPOU
FUNCTION_BLOCK YAHOO_WEATHER_ICON_OSCAT
VAR_IN_OUT
	YW : YAHOO_WEATHER_DATA;
END_VAR
VAR_INPUT
	ACTIVATE : BOOL;
END_VAR
VAR
	dat : ARRAY[0..48] OF INT := [4,2,2,4,17,1,3,1,2,2,2,2,2,3,3,3,3,5,3,6,7,14,8,9,9,10,9,11,12,11,12,13,14,15,16,4,14,4,17,2,2,3,3,3,12,2,3,4,0];
	act_last : BOOL;
	x : INT;
END_VAR

(*

version 1.0		04. may. 2011
programmer 		ks
tested by			ks

YAHOO_WEATHER_ICON_OSCAT ändert die ICON Nummer auf den OSCAT-Standard um
*)

IF ACTIVATE AND act_last = FALSE THEN
	x := MIN(YW.CUR_CONDITIONS_CODE,48);
	YW.CUR_CONDITIONS_ICON := dat[x];
	x := MIN(YW.FORCAST_TODAY_CODE,48);
	YW.FORCAST_TODAY_ICON := dat[x];
	x := MIN(YW.FORCAST_TOMORROW_CODE,48);
	YW.FORCAST_TOMORROW_ICON := dat[x];
END_IF;
act_last := ACTIVATE;

(* revision history
ks	04. may. 2011	rev 1.0
	original version
*)

END_FUNCTION_BLOCK

// ---- POUs/DRIVER/IRTRANS_RCV_1.TcPOU
FUNCTION_BLOCK IRTRANS_RCV_1
VAR_INPUT CONSTANT
	DEV_CODE : STRING;
	KEY_CODE : STRING;
END_VAR
VAR_INPUT
	CMD : BOOL;
END_VAR
VAR_IN_OUT
	DEV : STRING;
	KEY : STRING;
END_VAR
VAR_OUTPUT
	Q : BOOL;
END_VAR


(*

version 1.3	06. dec. 2009
programmer 	hugo
tested by		oscat

*)

Q := cmd AND dev_code = dev AND key_code = key;

(* revision history
hm	2. jan 2008		rev 1.0
	original version

hm	20. 6. 2008		rev 1.1
	performance improvement

hm	19. oct. 2008	rev 1.2
	changed input device_code to dev_code and device to dev for compatibility reasons

hm	06. dec. 2008	rev 1.3
	IRTRANS_1 renamed to IRTRANS_RCV_1

*)

END_FUNCTION_BLOCK

// ---- POUs/DRIVER/IRTRANS_RCV_8.TcPOU
FUNCTION_BLOCK IRTRANS_RCV_8
VAR_INPUT CONSTANT
	dev_code : STRING;
	key_code_0 : STRING;
	key_code_1 : STRING;
	key_code_2 : STRING;
	key_code_3 : STRING;
	key_code_4 : STRING;
	key_code_5 : STRING;
	key_code_6 : STRING;
	key_code_7 : STRING;
END_VAR
VAR_INPUT
	CMD : BOOL;
END_VAR
VAR_IN_OUT
	DEV : STRING;
	KEY : STRING;
END_VAR
VAR_OUTPUT
	Q0, Q1, Q2, Q3, Q4, Q5, Q6, Q7 : BOOL;
END_VAR
VAR_TEMP
	decode: BOOL;
END_VAR

(*

version 1.3	06. dec. 2009
programmer 	hugo
tested BY	oscat

*)

decode := cmd AND dev_code = dev;

Q0 := key = key_code_0 AND decode;
Q1 := key = key_code_1 AND decode;
Q2 := key = key_code_2 AND decode;
Q3 := key = key_code_3 AND decode;
Q4 := key = key_code_4 AND decode;
Q5 := key = key_code_5 AND decode;
Q6 := key = key_code_6 AND decode;
Q7 := key = key_code_7 AND decode;


(* revision history
hm	2. jan 2008		rev 1.0
	original version

hm	17. oct 2008	rev 1.1
	improved performance

hm	19. oct. 2008	rev 1.2
	changed input device_code to dev_code and device to dev for compatibility reasons

hm	06. dec. 2008	rev 1.3
	IRTRANS_1 renamed to IRTRANS_RCV_8

*)

END_FUNCTION_BLOCK

// ---- POUs/DRIVER/IRTRANS_SND_1.TcPOU
FUNCTION_BLOCK IRTRANS_SND_1
VAR_INPUT CONSTANT
	DEV_CODE : STRING;
	KEY_CODE : STRING;
END_VAR
VAR_INPUT
	IN : BOOL;
	T_REPEAT : TIME;
END_VAR
VAR_IN_OUT
	IP_C : IP_C; (* IP_Control Verwaltungsstruktur *)
	S_BUF : NETWORK_BUFFER_SHORT;
END_VAR
VAR_OUTPUT
	KEY : BYTE;
END_VAR
VAR
	skey : STRING;
	size : INT;
	str : STRING;
	t : TON;
	k : BYTE;
	lk : BYTE;
	d : BOOL;
END_VAR

(*
version 1.0		06. dec. 2009
programmer 		ks
tested by		ks
*)

d := IP_C.C_STATE > 127 AND (IP_C.MAILBOX[1] > 0 OR IP_C.C_MODE <> 5);
IF NOT d THEN RETURN; END_IF;

t(IN:= lk = k , PT:=T_REPEAT);

IF S_BUF.SIZE = 0 THEN
	IF IN THEN
		skey := KEY_CODE; k := 1;
	ELSE
		lk := 0;
		KEY := 0;
		RETURN; (* beenden wenn kein Key aktiv *)
	END_IF;

	IF lk <> k OR T.Q THEN (* anderer Key oder repeat wartezeit abgelaufen *)
		str := CONCAT('snd ',dev_code);
		str := CONCAT(str,',');
		str := CONCAT(str,skey);
		size := LEN(str);
		_STRING_TO_BUFFER(STR:=str, POS:=0, PT:=ADR(S_BUF.BUFFER), SIZE:=size);
		S_BUF.SIZE := size; (* Sendelänge eintragen *)
		KEY := k;
		lk := k; (* letzten Key speichern *)
		t(IN:=FALSE); (* Reset Time *)
	END_IF;
END_IF;

(* revision history
hm	6. dec 2009		rev 1.0
	original version
*)

END_FUNCTION_BLOCK

// ---- POUs/DRIVER/IRTRANS_SND_4.TcPOU
FUNCTION_BLOCK IRTRANS_SND_4
VAR_INPUT CONSTANT
	DEV_CODE : STRING;
	KEY_CODE_0 : STRING;
	KEY_CODE_1 : STRING;
	KEY_CODE_2 : STRING;
	KEY_CODE_3 : STRING;
END_VAR
VAR_INPUT
	IN_0 : BOOL;
	IN_1 : BOOL;
	IN_2 : BOOL;
	IN_3 : BOOL;
	T_REPEAT : TIME;
END_VAR
VAR_IN_OUT
	IP_C : IP_C; (* IP_Control Verwaltungsstruktur *)
	S_BUF : NETWORK_BUFFER_SHORT;
END_VAR
VAR_OUTPUT
	KEY : BYTE;
END_VAR
VAR
	skey : STRING;
	size : INT;
	str : STRING;
	t : TON;
	k : BYTE;
	lk : BYTE;
	d : BOOL;
END_VAR

(*
version 1.0		06. dec. 2009
programmer 		ks
tested by		ks
*)

d := IP_C.C_STATE > 127 AND (IP_C.MAILBOX[1] > 0 OR IP_C.C_MODE <> 5);
IF NOT d THEN RETURN; END_IF;

t(IN:= lk = k , PT:=T_REPEAT);

IF S_BUF.SIZE = 0 THEN
	IF IN_0 THEN
		skey := KEY_CODE_0; k := 1;
	ELSIF IN_1 THEN
		skey := KEY_CODE_1; k := 2;
	ELSIF IN_2 THEN
		skey := KEY_CODE_2; k := 3;
	ELSIF IN_3 THEN
		skey := KEY_CODE_3; k := 4;
	ELSE
		lk := 0;
		KEY := 0;
		RETURN; (* beenden wenn kein Key aktiv *)
	END_IF;

	IF lk <> k OR T.Q THEN (* anderer Key oder repeat wartezeit abgelaufen *)
		str := CONCAT('snd ',dev_code);
		str := CONCAT(str,',');
		str := CONCAT(str,skey);
		size := LEN(str);
		_STRING_TO_BUFFER(STR:=str, POS:=0, PT:=ADR(S_BUF.BUFFER), SIZE:=size);
		S_BUF.SIZE := size; (* Sendelänge eintragen *)
		KEY := k;
		lk := k; (* letzten Key speichern *)
		t(IN:=FALSE); (* Reset Time *)
	END_IF;
END_IF;

(* revision history
hm	6. dec 2009		rev 1.0
	original version
*)

END_FUNCTION_BLOCK

// ---- POUs/OTHER/NETWORK_VERSION.TcPOU
FUNCTION NETWORK_VERSION : DWORD
VAR_INPUT
	IN : BOOL;
END_VAR

(*
version 1.0	02. feb 2011
programmer 	kst
tested by		oscat

network_version returns the version number in dword format
110 is library version 1.10
if IN = true, the release date will be returned

*)

IF in THEN
	NETWORK_VERSION := DATE_TO_DWORD(D#2011-12-01);
ELSE
	NETWORK_VERSION := 121;
END_IF;

(* revision history
ks	2. feb 2011	rev 1.0
	original version

*)

END_FUNCTION

// ---- POUs/TELNET_VISION/TN_SC_READ_ATTR.TcPOU
FUNCTION_BLOCK TN_SC_READ_ATTR
VAR
	in_Offset : INT;
END_VAR
VAR_INPUT
	Iin_Y : INT;
	Iin_X : INT;
END_VAR
VAR_OUTPUT
	Oby_ATTR : BYTE;
END_VAR
VAR_IN_OUT
	Xus_TN_SCREEN : us_TN_SCREEN;
END_VAR

(*
version 1.0		10. mai 2010
programmer		ks
tested by		ks

TN_SC_READ_ATTR gibt den Farbcode einer Koordinate vom Bildschirm aus

*)

IF TN_SC_XY_ERROR(Iin_X,Iin_Y) THEN RETURN; END_IF;
in_Offset := (Iin_Y * 80) + Iin_X;
Oby_ATTR := Xus_TN_SCREEN.bya_COLOR[in_Offset]; (* Attribute auslesen *)

(* revision history
ks	10. mai. 2010	rev 1.0
	original version
*)

END_FUNCTION_BLOCK

// ---- POUs/TELNET_VISION/TN_SC_READ_CHAR.TcPOU
FUNCTION_BLOCK TN_SC_READ_CHAR
VAR
	in_Offset : INT;
END_VAR
VAR_INPUT
	Iin_Y : INT;
	Iin_X : INT;
END_VAR
VAR_OUTPUT
	Oby_CHAR : BYTE;
END_VAR
VAR_IN_OUT
	Xus_TN_SCREEN : us_TN_SCREEN;
END_VAR

(*
version 1.0		10. mai 2010
programmer		ks
tested by		ks

TN_SC_READ_CHAR gibt das Zeichen einer Koordinate vom Bildschirm aus
*)

IF TN_SC_XY_ERROR(Iin_X,Iin_Y) THEN RETURN; END_IF;
in_Offset := (Iin_Y * 80) + Iin_X;
Oby_CHAR := Xus_TN_SCREEN.bya_CHAR[in_Offset]; (* Charakter auslesen *)

(* revision history
ks	10. mai. 2010	rev 1.0
	original version
*)

END_FUNCTION_BLOCK

// ---- POUs/TELNET_VISION/TN_SC_WRITE_ATTR.TcPOU
FUNCTION_BLOCK TN_SC_WRITE_ATTR
VAR
	in_Offset : INT;
END_VAR
VAR_INPUT
	Iin_Y : INT;
	Iin_X : INT;
	Iby_ATTR : BYTE;
END_VAR
VAR_IN_OUT
	Xus_TN_SCREEN : us_TN_SCREEN;
END_VAR

(*
version 1.0		10. mai 2010
programmer		ks
tested by		ks

TN_SC_WRITE_ATTR ändert an der angegebenen Koordinate den Farbcode
*)

IF TN_SC_XY_ERROR(Iin_X,Iin_Y) THEN RETURN; END_IF;
in_Offset := (Iin_Y * 80) + Iin_X;
Xus_TN_SCREEN.bya_COLOR[in_Offset] := Iby_ATTR; (* Attribute schreiben *)

(* revision history
ks	10. mai. 2010	rev 1.0
	original version
*)

END_FUNCTION_BLOCK

// ---- POUs/TELNET_VISION/TN_SC_WRITE_CHAR.TcPOU
FUNCTION_BLOCK TN_SC_WRITE_CHAR
VAR
	in_Offset : INT;
END_VAR
VAR_INPUT
	Iin_Y : INT;
	Iin_X : INT;
	Iby_CHAR : BYTE;
END_VAR
VAR_IN_OUT
	Xus_TN_SCREEN : us_TN_SCREEN;
END_VAR

(*
version 1.0		10. mai 2010
programmer		ks
tested by		ks

TN_SC_WRITE_CHAR schreibt ein einzelnes Zeichen an die angegebenen Koordinate ohne den vorhandenen Farbcode zu ändern 
*)

IF TN_SC_XY_ERROR(Iin_X,Iin_Y) THEN RETURN; END_IF;
in_Offset := (Iin_Y * 80) + Iin_X;
Xus_TN_SCREEN.bya_CHAR[in_Offset] := Iby_CHAR; (* Charakter schreiben *)

(* revision history
ks	10. mai. 2010	rev 1.0
	original version
*)

END_FUNCTION_BLOCK

// ---- POUs/TELNET_VISION/TN_SC_WRITE_EOS.TcPOU
FUNCTION_BLOCK TN_SC_WRITE_EOS
VAR
	TN_SC_WRITE : TN_SC_WRITE;
END_VAR
VAR_INPUT
	Iby_ATTR : BYTE;
	Ist_STRING : STRING;
END_VAR
VAR_IN_OUT
	Xus_TN_SCREEN : us_TN_SCREEN;
END_VAR

(*
version 1.0		10. mai 2010
programmer		ks
tested by		ks

TN_SC_WRITE_EOS schreibt einem Text an das Ende des zuletzt geschreibene Texts 
*)

TN_SC_WRITE(Iin_Y := Xus_TN_SCREEN.in_EOS_Offset / 80, (* aktuelle Zeile ausrechnen *)
			Iin_X := Xus_TN_SCREEN.in_EOS_Offset MOD 80, (* aktuelle Spalte ausrechnen *)
			Iby_ATTR := Iby_ATTR,
			Ist_STRING := Ist_STRING,
			Xus_TN_SCREEN := Xus_TN_SCREEN);

(* revision history
ks	10. mai. 2010	rev 1.0
	original version
*)

END_FUNCTION_BLOCK

// ---- POUs/WEATHER/MOON_PHASE.TcPOU
FUNCTION_BLOCK MOON_PHASE
VAR_INPUT
	XDT : DT;
	SCALE : BYTE := 12;
	UPDATE : TIME := T#1h;
END_VAR
VAR_OUTPUT
	PHASE : BYTE;
END_VAR
VAR
	x : UDINT;
	last_dt : DT;
END_VAR

(*
version 1.0		15. may. 2011
programmer		ks
tested by			ks

MOON_PHASE berechnet die aktuelle Mondphase
*)

IF XDT - last_dt > UPDATE THEN
	x := (DT_TO_UDINT(XDT) - 603240) MOD 2551392;
	PHASE := UDINT_TO_BYTE(SCALE * x / 2551392) ;
	last_dt := XDT;
END_IF;

(* revision history
ks	15.may. 2011	rev 1.0
	original version

*)

END_FUNCTION_BLOCK

// ---- Project Information/F_GetCompany.TcPOU
// This function has been automatically generated from the project information.
{attribute 'signature_flag' := '1073741824'}
{attribute 'TcGenerated'}
{attribute 'no-analysis'}
FUNCTION F_GetCompany : WSTRING
VAR_INPUT
	
END_VAR

F_GetCompany := "Oscat";

END_FUNCTION

// ---- Project Information/F_GetTitle.TcPOU
// This function has been automatically generated from the project information.
{attribute 'signature_flag' := '1073741824'}
{attribute 'TcGenerated'}
{attribute 'no-analysis'}
FUNCTION F_GetTitle : WSTRING
VAR_INPUT
	
END_VAR

F_GetTitle := "Oscat_Network";

END_FUNCTION

// ---- Project Information/F_GetVersion.TcPOU
// This function has been automatically generated from the project information.
{attribute 'signature_flag' := '1073741824'}
{attribute 'TcGenerated'}
{attribute 'no-analysis'}
FUNCTION F_GetVersion : ST_LibVersion
VAR_INPUT
	
END_VAR

F_GetVersion.iMajor := 1;
F_GetVersion.iMinor := 2;
F_GetVersion.iBuild := 1;
F_GetVersion.iRevision := 0;

END_FUNCTION
